LIN {X 0,Y 569.864,Z 352.293,A -85,B 0,C 180,E1 27134.007,E2 27134.007} C_VEL
LIN {X 0,Y 571.953,Z 355.251,A -85,B 0,C 180,E1 27133.743,E2 27133.743} C_VEL
LIN {X 0,Y 584.357,Z 373.532,A -85,B 0,C 180,E1 27132.228,E2 27132.228} C_VEL
LIN {X 0,Y 595.034,Z 390.48,A -85,B 0,C 180,E1 27130.982,E2 27130.982} C_VEL
LIN {X 0,Y 605.418,Z 407.827,A -85,B 0,C 180,E1 27129.82,E2 27129.82} C_VEL
LIN {X 0,Y 601.344,Z 587.031,A -85,B 0,C 180,E1 27127.412,E2 27127.412} C_VEL
LIN {X 0,Y 600.399,Z 594.727,A -85,B 0,C 180,E1 27127.369,E2 27127.369} C_VEL
LIN {X 0,Y 595.054,Z 615.267,A -85,B 0,C 180,E1 27127.472,E2 27127.472} C_VEL
LIN {X 0,Y 594.323,Z 621.871,A -85,B 0,C 180,E1 27127.429,E2 27127.429} C_VEL
LIN {X 0,Y 591.491,Z 740.275,A -85,B 0,C 180,E1 27125.822,E2 27125.822} C_VEL
LIN {X 0,Y 590.199,Z 765.933,A -85,B 0,C 180,E1 27125.308,E2 27125.308} C_VEL
LIN {X 0,Y 588.778,Z 786.603,A -85,B 0,C 180,E1 27124.752,E2 27124.752} C_VEL
LIN {X 0,Y 586.911,Z 809.672,A -85,B 0,C 180,E1 27123.973,E2 27123.973} C_VEL
LIN {X 0,Y 584.739,Z 831.447,A -85,B 0,C 180,E1 27123.058,E2 27123.058} C_VEL
LIN {X 0,Y 582.598,Z 851.106,A -85,B 0,C 180,E1 27122.085,E2 27122.085} C_VEL
LIN {X 0,Y 579.921,Z 873.043,A -85,B 0,C 180,E1 27120.803,E2 27120.803} C_VEL
LIN {X 0,Y 577.554,Z 891.278,A -85,B 0,C 180,E1 27119.565,E2 27119.565} C_VEL
LIN {X 0,Y 574.708,Z 912.427,A -85,B 0,C 180,E1 27117.905,E2 27117.905} C_VEL
LIN {X 0,Y 572.362,Z 929.084,A -85,B 0,C 180,E1 27116.398,E2 27116.398} C_VEL
LIN {X 0,Y 569.881,Z 946.877,A -85,B 0,C 180,E1 27114.572,E2 27114.572} C_VEL
LIN {X 0,Y 567.593,Z 963.267,A -85,B 0,C 180,E1 27112.616,E2 27112.616} C_VEL
LIN {X 0,Y 565.641,Z 978.22,A -85,B 0,C 180,E1 27110.596,E2 27110.596} C_VEL
LIN {X 0,Y 563.908,Z 992.141,A -85,B 0,C 180,E1 27108.398,E2 27108.398} C_VEL
LIN {X 0,Y 562.601,Z 1004.328,A -85,B 0,C 180,E1 27106.202,E2 27106.202} C_VEL
LIN {X 0,Y 561.55,Z 1015.061,A -85,B 0,C 180,E1 27103.909,E2 27103.909} C_VEL
LIN {X 0,Y 560.865,Z 1023.83,A -85,B 0,C 180,E1 27101.726,E2 27101.726} C_VEL
LIN {X 0,Y 560.352,Z 1032.037,A -85,B 0,C 180,E1 27099.241,E2 27099.241} C_VEL
LIN {X 0,Y 560.1,Z 1037.791,A -85,B 0,C 180,E1 27097.076,E2 27097.076} C_VEL
LIN {X 0,Y 559.965,Z 1042.874,A -85,B 0,C 180,E1 27094.609,E2 27094.609} C_VEL
LIN {X 0,Y 559.925,Z 1046.117,A -85,B 0,C 180,E1 27092.252,E2 27092.252} C_VEL
LIN {X 0,Y 559.918,Z 1047.976,A -85,B 0,C 180,E1 27090,E2 27090} C_VEL
LIN {X 0,Y 559.896,Z 1048.458,A -85,B 0,C 180,E1 27087.441,E2 27087.441} C_VEL
LIN {X 0,Y 559.901,Z 1047.57,A -85,B 0,C 180,E1 27085.288,E2 27085.288} C_VEL
LIN {X 0,Y 559.937,Z 1045.192,A -85,B 0,C 180,E1 27082.819,E2 27082.819} C_VEL
LIN {X 0,Y 559.998,Z 1041.245,A -85,B 0,C 180,E1 27080.442,E2 27080.442} C_VEL
LIN {X 0,Y 560.165,Z 1036.402,A -85,B 0,C 180,E1 27078.259,E2 27078.259} C_VEL
LIN {X 0,Y 560.544,Z 1028.866,A -85,B 0,C 180,E1 27075.644,E2 27075.644} C_VEL
LIN {X 0,Y 561.057,Z 1021.218,A -85,B 0,C 180,E1 27073.497,E2 27073.497} C_VEL
LIN {X 0,Y 561.93,Z 1011.097,A -85,B 0,C 180,E1 27071.104,E2 27071.104} C_VEL
LIN {X 0,Y 562.978,Z 1000.415,A -85,B 0,C 180,E1 27068.976,E2 27068.976} C_VEL
LIN {X 0,Y 564.484,Z 987.53,A -85,B 0,C 180,E1 27066.734,E2 27066.734} C_VEL
LIN {X 0,Y 566.302,Z 973.067,A -85,B 0,C 180,E1 27064.593,E2 27064.593} C_VEL
LIN {X 0,Y 568.423,Z 957.461,A -85,B 0,C 180,E1 27062.557,E2 27062.557} C_VEL
LIN {X 0,Y 570.744,Z 940.758,A -85,B 0,C 180,E1 27060.682,E2 27060.682} C_VEL
LIN {X 0,Y 573.203,Z 923.555,A -85,B 0,C 180,E1 27058.971,E2 27058.971} C_VEL
LIN {X 0,Y 575.887,Z 904.313,A -85,B 0,C 180,E1 27057.318,E2 27057.318} C_VEL
LIN {X 0,Y 578.42,Z 885.955,A -85,B 0,C 180,E1 27055.938,E2 27055.938} C_VEL
LIN {X 0,Y 581.277,Z 863.847,A -85,B 0,C 180,E1 27054.51,E2 27054.51} C_VEL
LIN {X 0,Y 583.53,Z 844.808,A -85,B 0,C 180,E1 27053.457,E2 27053.457} C_VEL
LIN {X 0,Y 585.978,Z 822.583,A -85,B 0,C 180,E1 27052.409,E2 27052.409} C_VEL
LIN {X 0,Y 588.031,Z 800.135,A -85,B 0,C 180,E1 27051.543,E2 27051.543} C_VEL
LIN {X 0,Y 589.972,Z 776.277,A -85,B 0,C 180,E1 27050.802,E2 27050.802} C_VEL
LIN {X 0,Y 591.358,Z 753.251,A -85,B 0,C 180,E1 27050.269,E2 27050.269} C_VEL
LIN {X 0,Y 592.323,Z 730.378,A -85,B 0,C 180,E1 27049.878,E2 27049.878} C_VEL
LIN {X 0,Y 598.539,Z 477.791,A -85,B 0,C 180,E1 27046.449,E2 27046.449} C_VEL
LIN {X 0,Y 600.073,Z 410.838,A -85,B 0,C 180,E1 27045.512,E2 27045.512} C_VEL
LIN {X 0,Y 587.214,Z 389.608,A -85,B 0,C 180,E1 27043.955,E2 27043.955} C_VEL
LIN {X 0,Y 573.32,Z 368.918,A -85,B 0,C 180,E1 27042.18,E2 27042.18} C_VEL
LIN {X 0,Y 567.731,Z 361.268,A -85,B 0,C 180,E1 27041.435,E2 27041.435} C_VEL
LIN {X 0,Y 564.464,Z 356.623,A -85,B 0,C 180,E1 27040.985,E2 27040.985} C_VEL
LIN {X 0,Y 562.218,Z 353.874,A -85,B 0,C 180,E1 27040.679,E2 27040.679} C_VEL
LIN {X 0,Y 561.563,Z 351.979,A -85,B 0,C 180,E1 27040.534,E2 27040.534} C_VEL
LIN {X 0,Y 561.445,Z 351.25,A -85,B 0,C 180,E1 27040.411,E2 27040.411} C_VEL
LIN {X 0,Y 561.381,Z 351.276,A -85,B 0,C 180,E1 27037.235,E2 27037.235} C_VEL
LIN {X 0,Y 561.417,Z 351.281,A -85,B 0,C 180,E1 27033.906,E2 27033.906} C_VEL
LIN {X 0,Y 561.401,Z 351.292,A -85,B 0,C 180,E1 27030.742,E2 27030.742} C_VEL
LIN {X 0,Y 561.387,Z 351.299,A -85,B 0,C 180,E1 27027.357,E2 27027.357} C_VEL
LIN {X 0,Y 561.441,Z 351.289,A -85,B 0,C 180,E1 27024.181,E2 27024.181} C_VEL
LIN {X 0,Y 561.381,Z 351.291,A -85,B 0,C 180,E1 27020.978,E2 27020.978} C_VEL
LIN {X 0,Y 561.424,Z 351.283,A -85,B 0,C 180,E1 27017.731,E2 27017.731} C_VEL
LIN {X 0,Y 561.386,Z 351.293,A -85,B 0,C 180,E1 27014.65,E2 27014.65} C_VEL
LIN {X 0,Y 561.389,Z 351.296,A -85,B 0,C 180,E1 27011.195,E2 27011.195} C_VEL
LIN {X 0,Y 561.437,Z 351.298,A -85,B 0,C 180,E1 27007.985,E2 27007.985} C_VEL
LIN {X 0,Y 561.379,Z 351.292,A -85,B 0,C 180,E1 27004.802,E2 27004.802} C_VEL
LIN {X 0,Y 561.433,Z 351.279,A -85,B 0,C 180,E1 27001.531,E2 27001.531} C_VEL
LIN {X 0,Y 561.384,Z 351.301,A -85,B 0,C 180,E1 26998.469,E2 26998.469} C_VEL
LIN {X 0,Y 561.4,Z 351.299,A -85,B 0,C 180,E1 26995.096,E2 26995.096} C_VEL
LIN {X 0,Y 561.401,Z 351.285,A -85,B 0,C 180,E1 26992.014,E2 26992.014} C_VEL
LIN {X 0,Y 561.38,Z 351.281,A -85,B 0,C 180,E1 26988.701,E2 26988.701} C_VEL
LIN {X 0,Y 561.448,Z 351.281,A -85,B 0,C 180,E1 26985.457,E2 26985.457} C_VEL
LIN {X 0,Y 561.382,Z 351.3,A -85,B 0,C 180,E1 26982.267,E2 26982.267} C_VEL
LIN {X 0,Y 561.412,Z 351.298,A -85,B 0,C 180,E1 26978.948,E2 26978.948} C_VEL
LIN {X 0,Y 561.388,Z 351.287,A -85,B 0,C 180,E1 26975.929,E2 26975.929} C_VEL
LIN {X 0,Y 561.386,Z 351.288,A -85,B 0,C 180,E1 26972.498,E2 26972.498} C_VEL
LIN {X 0,Y 561.419,Z 351.3,A -85,B 0,C 180,E1 26969.497,E2 26969.497} C_VEL
LIN {X 0,Y 561.38,Z 351.303,A -85,B 0,C 180,E1 26966.24,E2 26966.24} C_VEL
LIN {X 0,Y 561.441,Z 351.299,A -85,B 0,C 180,E1 26962.99,E2 26962.99} C_VEL
LIN {X 0,Y 561.382,Z 351.304,A -85,B 0,C 180,E1 26959.827,E2 26959.827} C_VEL
LIN {X 0,Y 561.555,Z 352.203,A -85,B 0,C 180,E1 26959.648,E2 26959.648} C_VEL
LIN {X 0,Y 563.435,Z 356.303,A -85,B 0,C 180,E1 26958.957,E2 26958.957} C_VEL
LIN {X 0,Y 569.718,Z 370.71,A -85,B 0,C 180,E1 26956.667,E2 26956.667} C_VEL
LIN {X 0,Y 570.766,Z 373.125,A -85,B 0,C 180,E1 26956.352,E2 26956.352} C_VEL
LIN {X 0,Y 582.747,Z 391.401,A -85,B 0,C 180,E1 26954.789,E2 26954.789} C_VEL
LIN {X 0,Y 595.371,Z 412.407,A -85,B 0,C 180,E1 26953.225,E2 26953.225} C_VEL
LIN {X 0,Y 600.003,Z 420.961,A -85,B 0,C 180,E1 26952.664,E2 26952.664} C_VEL
LIN {X 0,Y 600.16,Z 425.019,A -85,B 0,C 180,E1 26952.585,E2 26952.585} C_VEL
LIN {X 0,Y 593.701,Z 685.414,A -85,B 0,C 180,E1 26949.041,E2 26949.041} C_VEL
LIN {X 0,Y 591.65,Z 766.034,A -85,B 0,C 180,E1 26947.933,E2 26947.933} C_VEL
LIN {X 0,Y 590.187,Z 791.581,A -85,B 0,C 180,E1 26947.422,E2 26947.422} C_VEL
LIN {X 0,Y 588.579,Z 813.335,A -85,B 0,C 180,E1 26946.836,E2 26946.836} C_VEL
LIN {X 0,Y 586.38,Z 838.196,A -85,B 0,C 180,E1 26945.975,E2 26945.975} C_VEL
LIN {X 0,Y 584.287,Z 858.471,A -85,B 0,C 180,E1 26945.114,E2 26945.114} C_VEL
LIN {X 0,Y 581.811,Z 880.444,A -85,B 0,C 180,E1 26944.014,E2 26944.014} C_VEL
LIN {X 0,Y 579.215,Z 901.047,A -85,B 0,C 180,E1 26942.785,E2 26942.785} C_VEL
LIN {X 0,Y 576.615,Z 921.114,A -85,B 0,C 180,E1 26941.411,E2 26941.411} C_VEL
LIN {X 0,Y 573.894,Z 941.134,A -85,B 0,C 180,E1 26939.812,E2 26939.812} C_VEL
LIN {X 0,Y 571.553,Z 958.312,A -85,B 0,C 180,E1 26938.252,E2 26938.252} C_VEL
LIN {X 0,Y 568.994,Z 977.194,A -85,B 0,C 180,E1 26936.285,E2 26936.285} C_VEL
LIN {X 0,Y 567.016,Z 992.376,A -85,B 0,C 180,E1 26934.482,E2 26934.482} C_VEL
LIN {X 0,Y 564.997,Z 1008.815,A -85,B 0,C 180,E1 26932.245,E2 26932.245} C_VEL
LIN {X 0,Y 563.613,Z 1020.97,A -85,B 0,C 180,E1 26930.348,E2 26930.348} C_VEL
LIN {X 0,Y 562.316,Z 1034.002,A -85,B 0,C 180,E1 26928.023,E2 26928.023} C_VEL
LIN {X 0,Y 561.398,Z 1044.512,A -85,B 0,C 180,E1 26925.813,E2 26925.813} C_VEL
LIN {X 0,Y 560.745,Z 1053.948,A -85,B 0,C 180,E1 26923.509,E2 26923.509} C_VEL
LIN {X 0,Y 560.304,Z 1061.89,A -85,B 0,C 180,E1 26921.112,E2 26921.112} C_VEL
LIN {X 0,Y 560.065,Z 1067.774,A -85,B 0,C 180,E1 26918.935,E2 26918.935} C_VEL
LIN {X 0,Y 559.949,Z 1073.035,A -85,B 0,C 180,E1 26916.356,E2 26916.356} C_VEL
LIN {X 0,Y 559.914,Z 1076.033,A -85,B 0,C 180,E1 26914.199,E2 26914.199} C_VEL
LIN {X 0,Y 559.904,Z 1077.913,A -85,B 0,C 180,E1 26911.944,E2 26911.944} C_VEL
LIN {X 0,Y 559.896,Z 1078.345,A -85,B 0,C 180,E1 26909.488,E2 26909.488} C_VEL
LIN {X 0,Y 559.907,Z 1077.429,A -85,B 0,C 180,E1 26907.339,E2 26907.339} C_VEL
LIN {X 0,Y 559.931,Z 1075.107,A -85,B 0,C 180,E1 26904.98,E2 26904.98} C_VEL
LIN {X 0,Y 559.984,Z 1070.929,A -85,B 0,C 180,E1 26902.51,E2 26902.51} C_VEL
LIN {X 0,Y 560.134,Z 1066.227,A -85,B 0,C 180,E1 26900.444,E2 26900.444} C_VEL
LIN {X 0,Y 560.464,Z 1058.71,A -85,B 0,C 180,E1 26897.866,E2 26897.866} C_VEL
LIN {X 0,Y 560.952,Z 1050.667,A -85,B 0,C 180,E1 26895.655,E2 26895.655} C_VEL
LIN {X 0,Y 561.76,Z 1040.359,A -85,B 0,C 180,E1 26893.257,E2 26893.257} C_VEL
LIN {X 0,Y 562.796,Z 1028.901,A -85,B 0,C 180,E1 26891.027,E2 26891.027} C_VEL
LIN {X 0,Y 564.22,Z 1015.654,A -85,B 0,C 180,E1 26888.775,E2 26888.775} C_VEL
LIN {X 0,Y 565.906,Z 1001.267,A -85,B 0,C 180,E1 26886.685,E2 26886.685} C_VEL
LIN {X 0,Y 567.913,Z 985.575,A -85,B 0,C 180,E1 26884.67,E2 26884.67} C_VEL
LIN {X 0,Y 570.192,Z 968.342,A -85,B 0,C 180,E1 26882.758,E2 26882.758} C_VEL
LIN {X 0,Y 572.443,Z 951.643,A -85,B 0,C 180,E1 26881.121,E2 26881.121} C_VEL
LIN {X 0,Y 575.208,Z 931.042,A -85,B 0,C 180,E1 26879.369,E2 26879.369} C_VEL
LIN {X 0,Y 577.627,Z 912.745,A -85,B 0,C 180,E1 26878.015,E2 26878.015} C_VEL
LIN {X 0,Y 580.49,Z 889.767,A -85,B 0,C 180,E1 26876.551,E2 26876.551} C_VEL
LIN {X 0,Y 582.689,Z 870.64,A -85,B 0,C 180,E1 26875.509,E2 26875.509} C_VEL
LIN {X 0,Y 585.179,Z 847.637,A -85,B 0,C 180,E1 26874.445,E2 26874.445} C_VEL
LIN {X 0,Y 587.18,Z 825.79,A -85,B 0,C 180,E1 26873.619,E2 26873.619} C_VEL
LIN {X 0,Y 589.127,Z 802.224,A -85,B 0,C 180,E1 26872.895,E2 26872.895} C_VEL
LIN {X 0,Y 590.595,Z 778.451,A -85,B 0,C 180,E1 26872.352,E2 26872.352} C_VEL
LIN {X 0,Y 591.556,Z 755.977,A -85,B 0,C 180,E1 26871.973,E2 26871.973} C_VEL
LIN {X 0,Y 597.259,Z 507.123,A -85,B 0,C 180,E1 26868.626,E2 26868.626} C_VEL
LIN {X 0,Y 599.18,Z 421.264,A -85,B 0,C 180,E1 26867.448,E2 26867.448} C_VEL
LIN {X 0,Y 598.222,Z 418.74,A -85,B 0,C 180,E1 26867.326,E2 26867.326} C_VEL
LIN {X 0,Y 584.047,Z 394.647,A -85,B 0,C 180,E1 26865.677,E2 26865.677} C_VEL
LIN {X 0,Y 570.279,Z 372.684,A -85,B 0,C 180,E1 26863.973,E2 26863.973} C_VEL
LIN {X 0,Y 564.417,Z 358.728,A -85,B 0,C 180,E1 26861.903,E2 26861.903} C_VEL
LIN {X 0,Y 561.425,Z 351.294,A -85,B 0,C 180,E1 26860.743,E2 26860.743} C_VEL
LIN {X 0,Y 561.384,Z 351.292,A -85,B 0,C 180,E1 26857.656,E2 26857.656} C_VEL
LIN {X 0,Y 561.388,Z 351.287,A -85,B 0,C 180,E1 26854.252,E2 26854.252} C_VEL
LIN {X 0,Y 561.409,Z 351.284,A -85,B 0,C 180,E1 26851.217,E2 26851.217} C_VEL
LIN {X 0,Y 561.381,Z 351.287,A -85,B 0,C 180,E1 26847.933,E2 26847.933} C_VEL
LIN {X 0,Y 561.443,Z 351.291,A -85,B 0,C 180,E1 26844.732,E2 26844.732} C_VEL
LIN {X 0,Y 561.38,Z 351.299,A -85,B 0,C 180,E1 26841.525,E2 26841.525} C_VEL
LIN {X 0,Y 561.414,Z 351.282,A -85,B 0,C 180,E1 26838.268,E2 26838.268} C_VEL
LIN {X 0,Y 561.395,Z 351.288,A -85,B 0,C 180,E1 26835.128,E2 26835.128} C_VEL
LIN {X 0,Y 561.389,Z 351.3,A -85,B 0,C 180,E1 26831.819,E2 26831.819} C_VEL
LIN {X 0,Y 561.435,Z 351.276,A -85,B 0,C 180,E1 26828.604,E2 26828.604} C_VEL
LIN {X 0,Y 561.379,Z 351.288,A -85,B 0,C 180,E1 26825.417,E2 26825.417} C_VEL
LIN {X 0,Y 561.432,Z 351.297,A -85,B 0,C 180,E1 26822.143,E2 26822.143} C_VEL
LIN {X 0,Y 561.381,Z 351.274,A -85,B 0,C 180,E1 26819.081,E2 26819.081} C_VEL
LIN {X 0,Y 561.399,Z 351.293,A -85,B 0,C 180,E1 26815.71,E2 26815.71} C_VEL
LIN {X 0,Y 561.405,Z 351.288,A -85,B 0,C 180,E1 26812.632,E2 26812.632} C_VEL
LIN {X 0,Y 561.382,Z 351.278,A -85,B 0,C 180,E1 26809.325,E2 26809.325} C_VEL
LIN {X 0,Y 561.45,Z 351.297,A -85,B 0,C 180,E1 26806.07,E2 26806.07} C_VEL
LIN {X 0,Y 561.382,Z 351.29,A -85,B 0,C 180,E1 26802.909,E2 26802.909} C_VEL
LIN {X 0,Y 561.424,Z 351.279,A -85,B 0,C 180,E1 26799.678,E2 26799.678} C_VEL
LIN {X 0,Y 561.392,Z 351.299,A -85,B 0,C 180,E1 26796.598,E2 26796.598} C_VEL
LIN {X 0,Y 561.393,Z 351.3,A -85,B 0,C 180,E1 26793.167,E2 26793.167} C_VEL
LIN {X 0,Y 561.425,Z 351.278,A -85,B 0,C 180,E1 26790.087,E2 26790.087} C_VEL
LIN {X 0,Y 561.382,Z 351.284,A -85,B 0,C 180,E1 26786.838,E2 26786.838} C_VEL
LIN {X 0,Y 561.44,Z 351.284,A -85,B 0,C 180,E1 26783.609,E2 26783.609} C_VEL
LIN {X 0,Y 561.385,Z 351.292,A -85,B 0,C 180,E1 26780.464,E2 26780.464} C_VEL
LIN {X 0,Y 561.413,Z 351.266,A -85,B 0,C 180,E1 26777.204,E2 26777.204} C_VEL
LIN {X 0,Y 561.416,Z 351.4,A -85,B 0,C 180,E1 26774.971,E2 26774.971} C_VEL
LIN {X 0,Y 561.764,Z 352.877,A -85,B 0,C 180,E1 26774.84,E2 26774.84} C_VEL
LIN {X 0,Y 563.667,Z 355.936,A -85,B 0,C 180,E1 26774.584,E2 26774.584} C_VEL
LIN {X 0,Y 565.182,Z 357.543,A -85,B 0,C 180,E1 26774.396,E2 26774.396} C_VEL
LIN {X 0,Y 567.902,Z 361.521,A -85,B 0,C 180,E1 26774.045,E2 26774.045} C_VEL
LIN {X 0,Y 579.907,Z 379.342,A -85,B 0,C 180,E1 26772.551,E2 26772.551} C_VEL
LIN {X 0,Y 590.434,Z 396.155,A -85,B 0,C 180,E1 26771.299,E2 26771.299} C_VEL
LIN {X 0,Y 599.337,Z 411.062,A -85,B 0,C 180,E1 26770.282,E2 26770.282} C_VEL
LIN {X 0,Y 594.323,Z 621.871,A -85,B 0,C 180,E1 26767.429,E2 26767.429} C_VEL
LIN {X 0,Y 593.377,Z 629.565,A -85,B 0,C 180,E1 26767.385,E2 26767.385} C_VEL
LIN {X 0,Y 588.018,Z 650.1,A -85,B 0,C 180,E1 26767.491,E2 26767.491} C_VEL
LIN {X 0,Y 587.273,Z 656.704,A -85,B 0,C 180,E1 26767.448,E2 26767.448} C_VEL
LIN {X 0,Y 585.108,Z 741.247,A -85,B 0,C 180,E1 26766.284,E2 26766.284} C_VEL
LIN {X 0,Y 583.771,Z 766.42,A -85,B 0,C 180,E1 26765.771,E2 26765.771} C_VEL
LIN {X 0,Y 582.282,Z 787.179,A -85,B 0,C 180,E1 26765.207,E2 26765.207} C_VEL
LIN {X 0,Y 580.17,Z 811.758,A -85,B 0,C 180,E1 26764.357,E2 26764.357} C_VEL
LIN {X 0,Y 578.055,Z 832.103,A -85,B 0,C 180,E1 26763.49,E2 26763.49} C_VEL
LIN {X 0,Y 575.616,Z 853.587,A -85,B 0,C 180,E1 26762.411,E2 26762.411} C_VEL
LIN {X 0,Y 572.808,Z 875.188,A -85,B 0,C 180,E1 26761.111,E2 26761.111} C_VEL
LIN {X 0,Y 570.082,Z 895.415,A -85,B 0,C 180,E1 26759.702,E2 26759.702} C_VEL
LIN {X 0,Y 567.3,Z 914.704,A -85,B 0,C 180,E1 26758.13,E2 26758.13} C_VEL
LIN {X 0,Y 564.872,Z 931.192,A -85,B 0,C 180,E1 26756.605,E2 26756.605} C_VEL
LIN {X 0,Y 562.083,Z 950.048,A -85,B 0,C 180,E1 26754.599,E2 26754.599} C_VEL
LIN {X 0,Y 559.944,Z 964.791,A -85,B 0,C 180,E1 26752.799,E2 26752.799} C_VEL
LIN {X 0,Y 557.643,Z 981.381,A -85,B 0,C 180,E1 26750.466,E2 26750.466} C_VEL
LIN {X 0,Y 556.042,Z 993.781,A -85,B 0,C 180,E1 26748.451,E2 26748.451} C_VEL
LIN {X 0,Y 554.51,Z 1007.231,A -85,B 0,C 180,E1 26745.908,E2 26745.908} C_VEL
LIN {X 0,Y 553.567,Z 1016.753,A -85,B 0,C 180,E1 26743.794,E2 26743.794} C_VEL
LIN {X 0,Y 552.795,Z 1026.378,A -85,B 0,C 180,E1 26741.265,E2 26741.265} C_VEL
LIN {X 0,Y 552.35,Z 1033.227,A -85,B 0,C 180,E1 26739.061,E2 26739.061} C_VEL
LIN {X 0,Y 552.085,Z 1039.323,A -85,B 0,C 180,E1 26736.656,E2 26736.656} C_VEL
LIN {X 0,Y 551.964,Z 1043.913,A -85,B 0,C 180,E1 26734.155,E2 26734.155} C_VEL
LIN {X 0,Y 551.926,Z 1046.697,A -85,B 0,C 180,E1 26731.973,E2 26731.973} C_VEL
LIN {X 0,Y 551.907,Z 1048.478,A -85,B 0,C 180,E1 26729.377,E2 26729.377} C_VEL
LIN {X 0,Y 551.906,Z 1048.598,A -85,B 0,C 180,E1 26727.092,E2 26727.092} C_VEL
LIN {X 0,Y 551.915,Z 1047.498,A -85,B 0,C 180,E1 26724.803,E2 26724.803} C_VEL
LIN {X 0,Y 551.945,Z 1044.574,A -85,B 0,C 180,E1 26722.191,E2 26722.191} C_VEL
LIN {X 0,Y 552.022,Z 1040.994,A -85,B 0,C 180,E1 26720.091,E2 26720.091} C_VEL
LIN {X 0,Y 552.247,Z 1035.536,A -85,B 0,C 180,E1 26717.664,E2 26717.664} C_VEL
LIN {X 0,Y 552.659,Z 1028.281,A -85,B 0,C 180,E1 26715.22,E2 26715.22} C_VEL
LIN {X 0,Y 553.283,Z 1020.145,A -85,B 0,C 180,E1 26712.943,E2 26712.943} C_VEL
LIN {X 0,Y 554.253,Z 1009.629,A -85,B 0,C 180,E1 26710.504,E2 26710.504} C_VEL
LIN {X 0,Y 555.467,Z 998.753,A -85,B 0,C 180,E1 26708.345,E2 26708.345} C_VEL
LIN {X 0,Y 557.208,Z 984.751,A -85,B 0,C 180,E1 26705.962,E2 26705.962} C_VEL
LIN {X 0,Y 559.009,Z 971.523,A -85,B 0,C 180,E1 26704.009,E2 26704.009} C_VEL
LIN {X 0,Y 561.449,Z 954.593,A -85,B 0,C 180,E1 26701.831,E2 26701.831} C_VEL
LIN {X 0,Y 563.739,Z 939.212,A -85,B 0,C 180,E1 26700.106,E2 26700.106} C_VEL
LIN {X 0,Y 566.545,Z 920.579,A -85,B 0,C 180,E1 26698.269,E2 26698.269} C_VEL
LIN {X 0,Y 569.193,Z 902.626,A -85,B 0,C 180,E1 26696.739,E2 26696.739} C_VEL
LIN {X 0,Y 572.136,Z 882.347,A -85,B 0,C 180,E1 26695.225,E2 26695.225} C_VEL
LIN {X 0,Y 574.829,Z 861.887,A -85,B 0,C 180,E1 26693.928,E2 26693.928} C_VEL
LIN {X 0,Y 577.425,Z 840.954,A -85,B 0,C 180,E1 26692.78,E2 26692.78} C_VEL
LIN {X 0,Y 579.913,Z 818.416,A -85,B 0,C 180,E1 26691.758,E2 26691.758} C_VEL
LIN {X 0,Y 581.859,Z 798.04,A -85,B 0,C 180,E1 26690.985,E2 26690.985} C_VEL
LIN {X 0,Y 583.902,Z 772.802,A -85,B 0,C 180,E1 26690.227,E2 26690.227} C_VEL
LIN {X 0,Y 585.175,Z 752.148,A -85,B 0,C 180,E1 26689.756,E2 26689.756} C_VEL
LIN {X 0,Y 586.212,Z 727.492,A -85,B 0,C 180,E1 26689.342,E2 26689.342} C_VEL
LIN {X 0,Y 592.735,Z 474.327,A -85,B 0,C 180,E1 26685.878,E2 26685.878} C_VEL
LIN {X 0,Y 594.185,Z 414.117,A -85,B 0,C 180,E1 26685.027,E2 26685.027} C_VEL
LIN {X 0,Y 580.889,Z 392.482,A -85,B 0,C 180,E1 26683.378,E2 26683.378} C_VEL
LIN {X 0,Y 568.738,Z 374.274,A -85,B 0,C 180,E1 26681.784,E2 26681.784} C_VEL
LIN {X 0,Y 563.794,Z 367.478,A -85,B 0,C 180,E1 26681.112,E2 26681.112} C_VEL
LIN {X 0,Y 560.388,Z 362.809,A -85,B 0,C 180,E1 26680.637,E2 26680.637} C_VEL
LIN {X 0,Y 557.686,Z 358.97,A -85,B 0,C 180,E1 26680.25,E2 26680.25} C_VEL
LIN {X 0,Y 556.886,Z 357.84,A -85,B 0,C 180,E1 26680.135,E2 26680.135} C_VEL
LIN {X 0,Y 554.43,Z 355.202,A -85,B 0,C 180,E1 26679.792,E2 26679.792} C_VEL
LIN {X 0,Y 553.443,Z 352.256,A -85,B 0,C 180,E1 26679.574,E2 26679.574} C_VEL
LIN {X 0,Y 553.49,Z 352.239,A -85,B 0,C 180,E1 26676.466,E2 26676.466} C_VEL
LIN {X 0,Y 553.443,Z 352.291,A -85,B 0,C 180,E1 26673.191,E2 26673.191} C_VEL
LIN {X 0,Y 553.484,Z 352.286,A -85,B 0,C 180,E1 26669.872,E2 26669.872} C_VEL
LIN {X 0,Y 553.454,Z 352.29,A -85,B 0,C 180,E1 26666.814,E2 26666.814} C_VEL
LIN {X 0,Y 553.452,Z 352.289,A -85,B 0,C 180,E1 26663.397,E2 26663.397} C_VEL
LIN {X 0,Y 553.488,Z 352.282,A -85,B 0,C 180,E1 26660.295,E2 26660.295} C_VEL
LIN {X 0,Y 553.441,Z 352.282,A -85,B 0,C 180,E1 26657.019,E2 26657.019} C_VEL
LIN {X 0,Y 553.5,Z 352.269,A -85,B 0,C 180,E1 26653.796,E2 26653.796} C_VEL
LIN {X 0,Y 553.446,Z 352.281,A -85,B 0,C 180,E1 26650.619,E2 26650.619} C_VEL
LIN {X 0,Y 553.451,Z 352.286,A -85,B 0,C 180,E1 26647.161,E2 26647.161} C_VEL
LIN {X 0,Y 553.492,Z 352.285,A -85,B 0,C 180,E1 26643.936,E2 26643.936} C_VEL
LIN {X 0,Y 553.439,Z 352.277,A -85,B 0,C 180,E1 26640.725,E2 26640.725} C_VEL
LIN {X 0,Y 553.494,Z 352.267,A -85,B 0,C 180,E1 26637.515,E2 26637.515} C_VEL
LIN {X 0,Y 553.448,Z 352.291,A -85,B 0,C 180,E1 26634.297,E2 26634.297} C_VEL
LIN {X 0,Y 553.449,Z 352.288,A -85,B 0,C 180,E1 26630.852,E2 26630.852} C_VEL
LIN {X 0,Y 553.498,Z 352.273,A -85,B 0,C 180,E1 26627.586,E2 26627.586} C_VEL
LIN {X 0,Y 553.439,Z 352.27,A -85,B 0,C 180,E1 26624.357,E2 26624.357} C_VEL
LIN {X 0,Y 553.485,Z 352.268,A -85,B 0,C 180,E1 26621.133,E2 26621.133} C_VEL
LIN {X 0,Y 553.453,Z 352.287,A -85,B 0,C 180,E1 26617.942,E2 26617.942} C_VEL
LIN {X 0,Y 553.447,Z 352.289,A -85,B 0,C 180,E1 26614.533,E2 26614.533} C_VEL
LIN {X 0,Y 553.509,Z 352.286,A -85,B 0,C 180,E1 26611.281,E2 26611.281} C_VEL
LIN {X 0,Y 553.44,Z 352.29,A -85,B 0,C 180,E1 26608.118,E2 26608.118} C_VEL
LIN {X 0,Y 553.483,Z 352.288,A -85,B 0,C 180,E1 26604.81,E2 26604.81} C_VEL
LIN {X 0,Y 553.454,Z 352.291,A -85,B 0,C 180,E1 26601.636,E2 26601.636} C_VEL
LIN {X 0,Y 553.479,Z 352.358,A -85,B 0,C 180,E1 26600.616,E2 26600.616} C_VEL
LIN {X 0,Y 554.665,Z 355.655,A -85,B 0,C 180,E1 26600.077,E2 26600.077} C_VEL
LIN {X 0,Y 558.806,Z 364.624,A -85,B 0,C 180,E1 26598.543,E2 26598.543} C_VEL
LIN {X 0,Y 562.281,Z 372.587,A -85,B 0,C 180,E1 26597.297,E2 26597.297} C_VEL
LIN {X 0,Y 574.651,Z 391.348,A -85,B 0,C 180,E1 26595.615,E2 26595.615} C_VEL
LIN {X 0,Y 587.888,Z 412.893,A -85,B 0,C 180,E1 26593.921,E2 26593.921} C_VEL
LIN {X 0,Y 594.346,Z 424.545,A -85,B 0,C 180,E1 26593.121,E2 26593.121} C_VEL
LIN {X 0,Y 587.538,Z 685.487,A -85,B 0,C 180,E1 26589.538,E2 26589.538} C_VEL
LIN {X 0,Y 585.395,Z 765.84,A -85,B 0,C 180,E1 26588.423,E2 26588.423} C_VEL
LIN {X 0,Y 583.856,Z 791.505,A -85,B 0,C 180,E1 26587.907,E2 26587.907} C_VEL
LIN {X 0,Y 582.157,Z 813.446,A -85,B 0,C 180,E1 26587.311,E2 26587.311} C_VEL
LIN {X 0,Y 579.857,Z 838.217,A -85,B 0,C 180,E1 26586.445,E2 26586.445} C_VEL
LIN {X 0,Y 577.731,Z 857.924,A -85,B 0,C 180,E1 26585.601,E2 26585.601} C_VEL
LIN {X 0,Y 575.077,Z 880.382,A -85,B 0,C 180,E1 26584.468,E2 26584.468} C_VEL
LIN {X 0,Y 572.309,Z 901.331,A -85,B 0,C 180,E1 26583.205,E2 26583.205} C_VEL
LIN {X 0,Y 569.514,Z 921.819,A -85,B 0,C 180,E1 26581.783,E2 26581.783} C_VEL
LIN {X 0,Y 566.635,Z 941.805,A -85,B 0,C 180,E1 26580.156,E2 26580.156} C_VEL
LIN {X 0,Y 564.042,Z 959.907,A -85,B 0,C 180,E1 26578.481,E2 26578.481} C_VEL
LIN {X 0,Y 561.436,Z 977.937,A -85,B 0,C 180,E1 26576.553,E2 26576.553} C_VEL
LIN {X 0,Y 559.365,Z 993.012,A -85,B 0,C 180,E1 26574.726,E2 26574.726} C_VEL
LIN {X 0,Y 557.245,Z 1009.251,A -85,B 0,C 180,E1 26572.468,E2 26572.468} C_VEL
LIN {X 0,Y 555.717,Z 1022.031,A -85,B 0,C 180,E1 26570.43,E2 26570.43} C_VEL
LIN {X 0,Y 554.313,Z 1035.345,A -85,B 0,C 180,E1 26567.966,E2 26567.966} C_VEL
LIN {X 0,Y 553.459,Z 1044.756,A -85,B 0,C 180,E1 26565.939,E2 26565.939} C_VEL
LIN {X 0,Y 552.749,Z 1054.477,A -85,B 0,C 180,E1 26563.495,E2 26563.495} C_VEL
LIN {X 0,Y 552.313,Z 1061.979,A -85,B 0,C 180,E1 26561.169,E2 26561.169} C_VEL
LIN {X 0,Y 552.061,Z 1068.073,A -85,B 0,C 180,E1 26558.856,E2 26558.856} C_VEL
LIN {X 0,Y 551.95,Z 1072.982,A -85,B 0,C 180,E1 26556.344,E2 26556.344} C_VEL
LIN {X 0,Y 551.916,Z 1075.818,A -85,B 0,C 180,E1 26554.26,E2 26554.26} C_VEL
LIN {X 0,Y 551.907,Z 1077.7,A -85,B 0,C 180,E1 26551.973,E2 26551.973} C_VEL
LIN {X 0,Y 551.899,Z 1078.132,A -85,B 0,C 180,E1 26549.481,E2 26549.481} C_VEL
LIN {X 0,Y 551.91,Z 1077.216,A -85,B 0,C 180,E1 26547.3,E2 26547.3} C_VEL
LIN {X 0,Y 551.933,Z 1074.893,A -85,B 0,C 180,E1 26544.907,E2 26544.907} C_VEL
LIN {X 0,Y 551.985,Z 1070.925,A -85,B 0,C 180,E1 26542.506,E2 26542.506} C_VEL
LIN {X 0,Y 552.143,Z 1066.011,A -85,B 0,C 180,E1 26540.304,E2 26540.304} C_VEL
LIN {X 0,Y 552.484,Z 1058.767,A -85,B 0,C 180,E1 26537.769,E2 26537.769} C_VEL
LIN {X 0,Y 552.991,Z 1050.86,A -85,B 0,C 180,E1 26535.551,E2 26535.551} C_VEL
LIN {X 0,Y 553.802,Z 1041.052,A -85,B 0,C 180,E1 26533.209,E2 26533.209} C_VEL
LIN {X 0,Y 554.932,Z 1029.263,A -85,B 0,C 180,E1 26530.857,E2 26530.857} C_VEL
LIN {X 0,Y 556.317,Z 1016.916,A -85,B 0,C 180,E1 26528.712,E2 26528.712} C_VEL
LIN {X 0,Y 558.197,Z 1001.827,A -85,B 0,C 180,E1 26526.456,E2 26526.456} C_VEL
LIN {X 0,Y 560.083,Z 987.69,A -85,B 0,C 180,E1 26524.601,E2 26524.601} C_VEL
LIN {X 0,Y 562.679,Z 969.137,A -85,B 0,C 180,E1 26522.482,E2 26522.482} C_VEL
LIN {X 0,Y 564.952,Z 953.042,A -85,B 0,C 180,E1 26520.875,E2 26520.875} C_VEL
LIN {X 0,Y 567.91,Z 932.216,A -85,B 0,C 180,E1 26519.062,E2 26519.062} C_VEL
LIN {X 0,Y 570.445,Z 913.895,A -85,B 0,C 180,E1 26517.682,E2 26517.682} C_VEL
LIN {X 0,Y 573.323,Z 892.216,A -85,B 0,C 180,E1 26516.263,E2 26516.263} C_VEL
LIN {X 0,Y 575.838,Z 871.262,A -85,B 0,C 180,E1 26515.1,E2 26515.1} C_VEL
LIN {X 0,Y 578.364,Z 849.264,A -85,B 0,C 180,E1 26514.06,E2 26514.06} C_VEL
LIN {X 0,Y 580.57,Z 826.283,A -85,B 0,C 180,E1 26513.177,E2 26513.177} C_VEL
LIN {X 0,Y 582.501,Z 803.812,A -85,B 0,C 180,E1 26512.475,E2 26512.475} C_VEL
LIN {X 0,Y 584.13,Z 779.377,A -85,B 0,C 180,E1 26511.9,E2 26511.9} C_VEL
LIN {X 0,Y 585.129,Z 757.488,A -85,B 0,C 180,E1 26511.522,E2 26511.522} C_VEL
LIN {X 0,Y 591.025,Z 513.048,A -85,B 0,C 180,E1 26508.202,E2 26508.202} C_VEL
LIN {X 0,Y 593.157,Z 423.688,A -85,B 0,C 180,E1 26506.968,E2 26506.968} C_VEL
LIN {X 0,Y 578.927,Z 399.379,A -85,B 0,C 180,E1 26505.276,E2 26505.276} C_VEL
LIN {X 0,Y 565.486,Z 377.953,A -85,B 0,C 180,E1 26503.581,E2 26503.581} C_VEL
LIN {X 0,Y 561.718,Z 372.03,A -85,B 0,C 180,E1 26503.052,E2 26503.052} C_VEL
LIN {X 0,Y 554.96,Z 356.032,A -85,B 0,C 180,E1 26500.574,E2 26500.574} C_VEL
LIN {X 0,Y 553.473,Z 352.517,A -85,B 0,C 180,E1 26500.005,E2 26500.005} C_VEL
LIN {X 0,Y 553.493,Z 352.272,A -85,B 0,C 180,E1 26497.112,E2 26497.112} C_VEL
LIN {X 0,Y 553.44,Z 352.278,A -85,B 0,C 180,E1 26493.811,E2 26493.811} C_VEL
LIN {X 0,Y 553.479,Z 352.271,A -85,B 0,C 180,E1 26490.507,E2 26490.507} C_VEL
LIN {X 0,Y 553.448,Z 352.27,A -85,B 0,C 180,E1 26487.432,E2 26487.432} C_VEL
LIN {X 0,Y 553.445,Z 352.273,A -85,B 0,C 180,E1 26483.985,E2 26483.985} C_VEL
LIN {X 0,Y 553.496,Z 352.286,A -85,B 0,C 180,E1 26480.848,E2 26480.848} C_VEL
LIN {X 0,Y 553.441,Z 352.287,A -85,B 0,C 180,E1 26477.561,E2 26477.561} C_VEL
LIN {X 0,Y 553.491,Z 352.264,A -85,B 0,C 180,E1 26474.329,E2 26474.329} C_VEL
LIN {X 0,Y 553.452,Z 352.286,A -85,B 0,C 180,E1 26471.146,E2 26471.146} C_VEL
LIN {X 0,Y 553.447,Z 352.29,A -85,B 0,C 180,E1 26467.683,E2 26467.683} C_VEL
LIN {X 0,Y 553.49,Z 352.262,A -85,B 0,C 180,E1 26464.559,E2 26464.559} C_VEL
LIN {X 0,Y 553.441,Z 352.288,A -85,B 0,C 180,E1 26461.346,E2 26461.346} C_VEL
LIN {X 0,Y 553.496,Z 352.266,A -85,B 0,C 180,E1 26458.137,E2 26458.137} C_VEL
LIN {X 0,Y 553.448,Z 352.277,A -85,B 0,C 180,E1 26454.921,E2 26454.921} C_VEL
LIN {X 0,Y 553.451,Z 352.29,A -85,B 0,C 180,E1 26451.481,E2 26451.481} C_VEL
LIN {X 0,Y 553.495,Z 352.26,A -85,B 0,C 180,E1 26448.221,E2 26448.221} C_VEL
LIN {X 0,Y 553.442,Z 352.281,A -85,B 0,C 180,E1 26445.027,E2 26445.027} C_VEL
LIN {X 0,Y 553.493,Z 352.285,A -85,B 0,C 180,E1 26441.788,E2 26441.788} C_VEL
LIN {X 0,Y 553.452,Z 352.269,A -85,B 0,C 180,E1 26438.596,E2 26438.596} C_VEL
LIN {X 0,Y 553.453,Z 352.27,A -85,B 0,C 180,E1 26435.22,E2 26435.22} C_VEL
LIN {X 0,Y 553.502,Z 352.284,A -85,B 0,C 180,E1 26431.986,E2 26431.986} C_VEL
LIN {X 0,Y 553.446,Z 352.29,A -85,B 0,C 180,E1 26428.767,E2 26428.767} C_VEL
LIN {X 0,Y 553.487,Z 352.281,A -85,B 0,C 180,E1 26425.465,E2 26425.465} C_VEL
LIN {X 0,Y 553.461,Z 352.285,A -85,B 0,C 180,E1 26422.233,E2 26422.233} C_VEL
LIN {X 0,Y 553.453,Z 352.292,A -85,B 0,C 180,E1 26418.881,E2 26418.881} C_VEL
LIN {X 0,Y 553.516,Z 352.422,A -85,B 0,C 180,E1 26415.747,E2 26415.747} C_VEL
LIN {X 0,Y 554.737,Z 355.613,A -85,B 0,C 180,E1 26415.552,E2 26415.552} C_VEL
LIN {X 0,Y 557.304,Z 358.568,A -85,B 0,C 180,E1 26415.216,E2 26415.216} C_VEL
LIN {X 0,Y 560.041,Z 362.58,A -85,B 0,C 180,E1 26414.848,E2 26414.848} C_VEL
LIN {X 0,Y 567.608,Z 373.212,A -85,B 0,C 180,E1 26413.868,E2 26413.868} C_VEL
LIN {X 0,Y 581.618,Z 394.667,A -85,B 0,C 180,E1 26412.132,E2 26412.132} C_VEL
LIN {X 0,Y 593.291,Z 414.33,A -85,B 0,C 180,E1 26410.753,E2 26410.753} C_VEL
LIN {X 0,Y 587.273,Z 656.704,A -85,B 0,C 180,E1 26407.448,E2 26407.448} C_VEL
LIN {X 0,Y 586.31,Z 664.399,A -85,B 0,C 180,E1 26407.405,E2 26407.405} C_VEL
LIN {X 0,Y 580.934,Z 684.929,A -85,B 0,C 180,E1 26407.514,E2 26407.514} C_VEL
LIN {X 0,Y 580.191,Z 691.532,A -85,B 0,C 180,E1 26407.47,E2 26407.47} C_VEL
LIN {X 0,Y 578.713,Z 743.986,A -85,B 0,C 180,E1 26406.727,E2 26406.727} C_VEL
LIN {X 0,Y 577.312,Z 767.92,A -85,B 0,C 180,E1 26406.219,E2 26406.219} C_VEL
LIN {X 0,Y 575.729,Z 789.042,A -85,B 0,C 180,E1 26405.633,E2 26405.633} C_VEL
LIN {X 0,Y 573.476,Z 813.615,A -85,B 0,C 180,E1 26404.76,E2 26404.76} C_VEL
LIN {X 0,Y 571.275,Z 833.863,A -85,B 0,C 180,E1 26403.88,E2 26403.88} C_VEL
LIN {X 0,Y 568.599,Z 856.085,A -85,B 0,C 180,E1 26402.734,E2 26402.734} C_VEL
LIN {X 0,Y 565.934,Z 875.723,A -85,B 0,C 180,E1 26401.532,E2 26401.532} C_VEL
LIN {X 0,Y 562.986,Z 896.638,A -85,B 0,C 180,E1 26400.056,E2 26400.056} C_VEL
LIN {X 0,Y 560.079,Z 915.772,A -85,B 0,C 180,E1 26398.468,E2 26398.468} C_VEL
LIN {X 0,Y 557.469,Z 932.739,A -85,B 0,C 180,E1 26396.872,E2 26396.872} C_VEL
LIN {X 0,Y 554.693,Z 950.508,A -85,B 0,C 180,E1 26394.945,E2 26394.945} C_VEL
LIN {X 0,Y 552.453,Z 965.214,A -85,B 0,C 180,E1 26393.126,E2 26393.126} C_VEL
LIN {X 0,Y 550.12,Z 981.104,A -85,B 0,C 180,E1 26390.87,E2 26390.87} C_VEL
LIN {X 0,Y 548.462,Z 993.237,A -85,B 0,C 180,E1 26388.882,E2 26388.882} C_VEL
LIN {X 0,Y 546.884,Z 1006.084,A -85,B 0,C 180,E1 26386.463,E2 26386.463} C_VEL
LIN {X 0,Y 545.776,Z 1016.202,A -85,B 0,C 180,E1 26384.211,E2 26384.211} C_VEL
LIN {X 0,Y 544.95,Z 1025.658,A -85,B 0,C 180,E1 26381.751,E2 26381.751} C_VEL
LIN {X 0,Y 544.408,Z 1033.231,A -85,B 0,C 180,E1 26379.301,E2 26379.301} C_VEL
LIN {X 0,Y 544.119,Z 1039.11,A -85,B 0,C 180,E1 26376.966,E2 26376.966} C_VEL
LIN {X 0,Y 543.975,Z 1043.859,A -85,B 0,C 180,E1 26374.428,E2 26374.428} C_VEL
LIN {X 0,Y 543.935,Z 1046.719,A -85,B 0,C 180,E1 26372.212,E2 26372.212} C_VEL
LIN {X 0,Y 543.91,Z 1048.63,A -85,B 0,C 180,E1 26369.684,E2 26369.684} C_VEL
LIN {X 0,Y 543.904,Z 1048.85,A -85,B 0,C 180,E1 26367.26,E2 26367.26} C_VEL
LIN {X 0,Y 543.911,Z 1047.945,A -85,B 0,C 180,E1 26365.125,E2 26365.125} C_VEL
LIN {X 0,Y 543.943,Z 1045.533,A -85,B 0,C 180,E1 26362.607,E2 26362.607} C_VEL
LIN {X 0,Y 544.029,Z 1041.559,A -85,B 0,C 180,E1 26360.158,E2 26360.158} C_VEL
LIN {X 0,Y 544.229,Z 1036.691,A -85,B 0,C 180,E1 26357.91,E2 26357.91} C_VEL
LIN {X 0,Y 544.667,Z 1029.45,A -85,B 0,C 180,E1 26355.325,E2 26355.325} C_VEL
LIN {X 0,Y 545.249,Z 1021.983,A -85,B 0,C 180,E1 26353.157,E2 26353.157} C_VEL
LIN {X 0,Y 546.21,Z 1012.263,A -85,B 0,C 180,E1 26350.761,E2 26350.761} C_VEL
LIN {X 0,Y 547.47,Z 1001.093,A -85,B 0,C 180,E1 26348.463,E2 26348.463} C_VEL
LIN {X 0,Y 549.156,Z 988.247,A -85,B 0,C 180,E1 26346.158,E2 26346.158} C_VEL
LIN {X 0,Y 551.198,Z 973.856,A -85,B 0,C 180,E1 26343.96,E2 26343.96} C_VEL
LIN {X 0,Y 553.43,Z 959.175,A -85,B 0,C 180,E1 26341.982,E2 26341.982} C_VEL
LIN {X 0,Y 556.081,Z 942.25,A -85,B 0,C 180,E1 26340.008,E2 26340.008} C_VEL
LIN {X 0,Y 558.6,Z 926.284,A -85,B 0,C 180,E1 26338.368,E2 26338.368} C_VEL
LIN {X 0,Y 561.851,Z 905.525,A -85,B 0,C 180,E1 26336.517,E2 26336.517} C_VEL
LIN {X 0,Y 564.509,Z 887.997,A -85,B 0,C 180,E1 26335.164,E2 26335.164} C_VEL
LIN {X 0,Y 567.634,Z 866.271,A -85,B 0,C 180,E1 26333.711,E2 26333.711} C_VEL
LIN {X 0,Y 570.163,Z 846.787,A -85,B 0,C 180,E1 26332.601,E2 26332.601} C_VEL
LIN {X 0,Y 572.736,Z 825.719,A -85,B 0,C 180,E1 26331.574,E2 26331.574} C_VEL
LIN {X 0,Y 575.102,Z 802.41,A -85,B 0,C 180,E1 26330.642,E2 26330.642} C_VEL
LIN {X 0,Y 577.063,Z 780.294,A -85,B 0,C 180,E1 26329.927,E2 26329.927} C_VEL
LIN {X 0,Y 578.78,Z 755.543,A -85,B 0,C 180,E1 26329.321,E2 26329.321} C_VEL
LIN {X 0,Y 579.816,Z 733.707,A -85,B 0,C 180,E1 26328.932,E2 26328.932} C_VEL
LIN {X 0,Y 586.618,Z 484.146,A -85,B 0,C 180,E1 26325.48,E2 26325.48} C_VEL
LIN {X 0,Y 588.402,Z 417.526,A -85,B 0,C 180,E1 26324.54,E2 26324.54} C_VEL
LIN {X 0,Y 575.019,Z 395.806,A -85,B 0,C 180,E1 26322.836,E2 26322.836} C_VEL
LIN {X 0,Y 561.085,Z 375.029,A -85,B 0,C 180,E1 26320.947,E2 26320.947} C_VEL
LIN {X 0,Y 553.737,Z 365.162,A -85,B 0,C 180,E1 26319.903,E2 26319.903} C_VEL
LIN {X 0,Y 550.099,Z 360.585,A -85,B 0,C 180,E1 26319.373,E2 26319.373} C_VEL
LIN {X 0,Y 549.271,Z 359.092,A -85,B 0,C 180,E1 26319.242,E2 26319.242} C_VEL
LIN {X 0,Y 546.699,Z 356.549,A -85,B 0,C 180,E1 26318.871,E2 26318.871} C_VEL
LIN {X 0,Y 545.557,Z 353.379,A -85,B 0,C 180,E1 26318.663,E2 26318.663} C_VEL
LIN {X 0,Y 545.5,Z 353.228,A -85,B 0,C 180,E1 26315.346,E2 26315.346} C_VEL
LIN {X 0,Y 545.56,Z 353.263,A -85,B 0,C 180,E1 26312.107,E2 26312.107} C_VEL
LIN {X 0,Y 545.51,Z 353.27,A -85,B 0,C 180,E1 26308.94,E2 26308.94} C_VEL
LIN {X 0,Y 545.517,Z 353.264,A -85,B 0,C 180,E1 26305.514,E2 26305.514} C_VEL
LIN {X 0,Y 545.558,Z 353.262,A -85,B 0,C 180,E1 26302.248,E2 26302.248} C_VEL
LIN {X 0,Y 545.507,Z 353.276,A -85,B 0,C 180,E1 26298.949,E2 26298.949} C_VEL
LIN {X 0,Y 545.541,Z 353.274,A -85,B 0,C 180,E1 26295.63,E2 26295.63} C_VEL
LIN {X 0,Y 545.517,Z 353.274,A -85,B 0,C 180,E1 26292.491,E2 26292.491} C_VEL
LIN {X 0,Y 545.506,Z 353.269,A -85,B 0,C 180,E1 26289.07,E2 26289.07} C_VEL
LIN {X 0,Y 545.561,Z 353.256,A -85,B 0,C 180,E1 26285.891,E2 26285.891} C_VEL
LIN {X 0,Y 545.504,Z 353.277,A -85,B 0,C 180,E1 26282.606,E2 26282.606} C_VEL
LIN {X 0,Y 545.533,Z 353.276,A -85,B 0,C 180,E1 26279.265,E2 26279.265} C_VEL
LIN {X 0,Y 545.532,Z 353.266,A -85,B 0,C 180,E1 26276.006,E2 26276.006} C_VEL
LIN {X 0,Y 545.502,Z 353.258,A -85,B 0,C 180,E1 26272.734,E2 26272.734} C_VEL
LIN {X 0,Y 545.559,Z 353.259,A -85,B 0,C 180,E1 26269.546,E2 26269.546} C_VEL
LIN {X 0,Y 545.504,Z 353.279,A -85,B 0,C 180,E1 26266.281,E2 26266.281} C_VEL
LIN {X 0,Y 545.528,Z 353.275,A -85,B 0,C 180,E1 26262.947,E2 26262.947} C_VEL
LIN {X 0,Y 545.531,Z 353.26,A -85,B 0,C 180,E1 26259.732,E2 26259.732} C_VEL
LIN {X 0,Y 545.502,Z 353.26,A -85,B 0,C 180,E1 26256.447,E2 26256.447} C_VEL
LIN {X 0,Y 545.562,Z 353.256,A -85,B 0,C 180,E1 26253.197,E2 26253.197} C_VEL
LIN {X 0,Y 545.503,Z 353.277,A -85,B 0,C 180,E1 26250.095,E2 26250.095} C_VEL
LIN {X 0,Y 545.538,Z 353.275,A -85,B 0,C 180,E1 26246.768,E2 26246.768} C_VEL
LIN {X 0,Y 545.522,Z 353.277,A -85,B 0,C 180,E1 26243.568,E2 26243.568} C_VEL
LIN {X 0,Y 545.547,Z 353.434,A -85,B 0,C 180,E1 26241.501,E2 26241.501} C_VEL
LIN {X 0,Y 546.943,Z 356.866,A -85,B 0,C 180,E1 26240.897,E2 26240.897} C_VEL
LIN {X 0,Y 552.731,Z 369.791,A -85,B 0,C 180,E1 26238.654,E2 26238.654} C_VEL
LIN {X 0,Y 553.923,Z 372.421,A -85,B 0,C 180,E1 26238.269,E2 26238.269} C_VEL
LIN {X 0,Y 566.29,Z 390.72,A -85,B 0,C 180,E1 26236.517,E2 26236.517} C_VEL
LIN {X 0,Y 578.478,Z 410.325,A -85,B 0,C 180,E1 26234.89,E2 26234.89} C_VEL
LIN {X 0,Y 588.478,Z 427.51,A -85,B 0,C 180,E1 26233.62,E2 26233.62} C_VEL
LIN {X 0,Y 581.414,Z 685.931,A -85,B 0,C 180,E1 26230.041,E2 26230.041} C_VEL
LIN {X 0,Y 579.185,Z 765.672,A -85,B 0,C 180,E1 26228.924,E2 26228.924} C_VEL
LIN {X 0,Y 577.58,Z 791.315,A -85,B 0,C 180,E1 26228.405,E2 26228.405} C_VEL
LIN {X 0,Y 575.8,Z 813.335,A -85,B 0,C 180,E1 26227.803,E2 26227.803} C_VEL
LIN {X 0,Y 573.376,Z 838.25,A -85,B 0,C 180,E1 26226.924,E2 26226.924} C_VEL
LIN {X 0,Y 571.195,Z 857.607,A -85,B 0,C 180,E1 26226.09,E2 26226.09} C_VEL
LIN {X 0,Y 568.389,Z 880.253,A -85,B 0,C 180,E1 26224.938,E2 26224.938} C_VEL
LIN {X 0,Y 565.532,Z 900.948,A -85,B 0,C 180,E1 26223.678,E2 26223.678} C_VEL
LIN {X 0,Y 562.652,Z 920.988,A -85,B 0,C 180,E1 26222.277,E2 26222.277} C_VEL
LIN {X 0,Y 559.666,Z 940.68,A -85,B 0,C 180,E1 26220.668,E2 26220.668} C_VEL
LIN {X 0,Y 557.039,Z 958.054,A -85,B 0,C 180,E1 26219.053,E2 26219.053} C_VEL
LIN {X 0,Y 554.171,Z 976.838,A -85,B 0,C 180,E1 26217.045,E2 26217.045} C_VEL
LIN {X 0,Y 551.96,Z 991.974,A -85,B 0,C 180,E1 26215.196,E2 26215.196} C_VEL
LIN {X 0,Y 549.686,Z 1008.315,A -85,B 0,C 180,E1 26212.909,E2 26212.909} C_VEL
LIN {X 0,Y 548.05,Z 1021.164,A -85,B 0,C 180,E1 26210.841,E2 26210.841} C_VEL
LIN {X 0,Y 546.494,Z 1034.945,A -85,B 0,C 180,E1 26208.27,E2 26208.27} C_VEL
LIN {X 0,Y 545.565,Z 1044.534,A -85,B 0,C 180,E1 26206.175,E2 26206.175} C_VEL
LIN {X 0,Y 544.805,Z 1054.257,A -85,B 0,C 180,E1 26203.695,E2 26203.695} C_VEL
LIN {X 0,Y 544.338,Z 1061.76,A -85,B 0,C 180,E1 26201.335,E2 26201.335} C_VEL
LIN {X 0,Y 544.07,Z 1067.856,A -85,B 0,C 180,E1 26198.987,E2 26198.987} C_VEL
LIN {X 0,Y 543.949,Z 1072.766,A -85,B 0,C 180,E1 26196.438,E2 26196.438} C_VEL
LIN {X 0,Y 543.918,Z 1075.604,A -85,B 0,C 180,E1 26194.323,E2 26194.323} C_VEL
LIN {X 0,Y 543.91,Z 1077.486,A -85,B 0,C 180,E1 26192.002,E2 26192.002} C_VEL
LIN {X 0,Y 543.902,Z 1077.918,A -85,B 0,C 180,E1 26189.473,E2 26189.473} C_VEL
LIN {X 0,Y 543.912,Z 1077.003,A -85,B 0,C 180,E1 26187.26,E2 26187.26} C_VEL
LIN {X 0,Y 543.934,Z 1074.679,A -85,B 0,C 180,E1 26184.832,E2 26184.832} C_VEL
LIN {X 0,Y 543.986,Z 1070.71,A -85,B 0,C 180,E1 26182.395,E2 26182.395} C_VEL
LIN {X 0,Y 544.145,Z 1066.055,A -85,B 0,C 180,E1 26180.267,E2 26180.267} C_VEL
LIN {X 0,Y 544.484,Z 1059.287,A -85,B 0,C 180,E1 26177.808,E2 26177.808} C_VEL
LIN {X 0,Y 545.031,Z 1051.054,A -85,B 0,C 180,E1 26175.444,E2 26175.444} C_VEL
LIN {X 0,Y 545.787,Z 1042.23,A -85,B 0,C 180,E1 26173.284,E2 26173.284} C_VEL
LIN {X 0,Y 547.007,Z 1030.206,A -85,B 0,C 180,E1 26170.79,E2 26170.79} C_VEL
LIN {X 0,Y 548.367,Z 1018.548,A -85,B 0,C 180,E1 26168.711,E2 26168.711} C_VEL
LIN {X 0,Y 550.294,Z 1003.93,A -85,B 0,C 180,E1 26166.438,E2 26166.438} C_VEL
LIN {X 0,Y 552.309,Z 989.361,A -85,B 0,C 180,E1 26164.477,E2 26164.477} C_VEL
LIN {X 0,Y 554.838,Z 972.333,A -85,B 0,C 180,E1 26162.456,E2 26162.456} C_VEL
LIN {X 0,Y 557.462,Z 954.481,A -85,B 0,C 180,E1 26160.628,E2 26160.628} C_VEL
LIN {X 0,Y 560.362,Z 935.264,A -85,B 0,C 180,E1 26158.897,E2 26158.897} C_VEL
LIN {X 0,Y 563.173,Z 915.778,A -85,B 0,C 180,E1 26157.395,E2 26157.395} C_VEL
LIN {X 0,Y 565.83,Z 896.882,A -85,B 0,C 180,E1 26156.115,E2 26156.115} C_VEL
LIN {X 0,Y 568.774,Z 873.901,A -85,B 0,C 180,E1 26154.787,E2 26154.787} C_VEL
LIN {X 0,Y 571.274,Z 853.014,A -85,B 0,C 180,E1 26153.77,E2 26153.77} C_VEL
LIN {X 0,Y 573.845,Z 828.285,A -85,B 0,C 180,E1 26152.778,E2 26152.778} C_VEL
LIN {X 0,Y 575.738,Z 807.183,A -85,B 0,C 180,E1 26152.098,E2 26152.098} C_VEL
LIN {X 0,Y 577.644,Z 781.289,A -85,B 0,C 180,E1 26151.458,E2 26151.458} C_VEL
LIN {X 0,Y 578.728,Z 759.201,A -85,B 0,C 180,E1 26151.065,E2 26151.065} C_VEL
LIN {X 0,Y 584.791,Z 520.135,A -85,B 0,C 180,E1 26147.786,E2 26147.786} C_VEL
LIN {X 0,Y 587.154,Z 426.916,A -85,B 0,C 180,E1 26146.489,E2 26146.489} C_VEL
LIN {X 0,Y 571.809,Z 400.651,A -85,B 0,C 180,E1 26144.612,E2 26144.612} C_VEL
LIN {X 0,Y 559.047,Z 380.64,A -85,B 0,C 180,E1 26142.957,E2 26142.957} C_VEL
LIN {X 0,Y 553.395,Z 371.842,A -85,B 0,C 180,E1 26142.163,E2 26142.163} C_VEL
LIN {X 0,Y 548.431,Z 360.447,A -85,B 0,C 180,E1 26140.333,E2 26140.333} C_VEL
LIN {X 0,Y 545.613,Z 353.686,A -85,B 0,C 180,E1 26139.216,E2 26139.216} C_VEL
LIN {X 0,Y 545.563,Z 353.268,A -85,B 0,C 180,E1 26139.085,E2 26139.085} C_VEL
LIN {X 0,Y 545.503,Z 353.282,A -85,B 0,C 180,E1 26135.783,E2 26135.783} C_VEL
LIN {X 0,Y 545.533,Z 353.276,A -85,B 0,C 180,E1 26132.482,E2 26132.482} C_VEL
LIN {X 0,Y 545.517,Z 353.275,A -85,B 0,C 180,E1 26129.421,E2 26129.421} C_VEL
LIN {X 0,Y 545.507,Z 353.274,A -85,B 0,C 180,E1 26125.981,E2 26125.981} C_VEL
LIN {X 0,Y 545.567,Z 353.251,A -85,B 0,C 180,E1 26122.75,E2 26122.75} C_VEL
LIN {X 0,Y 545.502,Z 353.261,A -85,B 0,C 180,E1 26119.488,E2 26119.488} C_VEL
LIN {X 0,Y 545.531,Z 353.274,A -85,B 0,C 180,E1 26116.173,E2 26116.173} C_VEL
LIN {X 0,Y 545.522,Z 353.268,A -85,B 0,C 180,E1 26113.029,E2 26113.029} C_VEL
LIN {X 0,Y 545.505,Z 353.253,A -85,B 0,C 180,E1 26109.708,E2 26109.708} C_VEL
LIN {X 0,Y 545.571,Z 353.272,A -85,B 0,C 180,E1 26106.419,E2 26106.419} C_VEL
LIN {X 0,Y 545.505,Z 353.27,A -85,B 0,C 180,E1 26103.152,E2 26103.152} C_VEL
LIN {X 0,Y 545.521,Z 353.252,A -85,B 0,C 180,E1 26099.79,E2 26099.79} C_VEL
LIN {X 0,Y 545.534,Z 353.275,A -85,B 0,C 180,E1 26096.638,E2 26096.638} C_VEL
LIN {X 0,Y 545.504,Z 353.259,A -85,B 0,C 180,E1 26093.369,E2 26093.369} C_VEL
LIN {X 0,Y 545.561,Z 353.262,A -85,B 0,C 180,E1 26090.186,E2 26090.186} C_VEL
LIN {X 0,Y 545.509,Z 353.276,A -85,B 0,C 180,E1 26086.863,E2 26086.863} C_VEL
LIN {X 0,Y 545.519,Z 353.257,A -85,B 0,C 180,E1 26083.459,E2 26083.459} C_VEL
LIN {X 0,Y 545.545,Z 353.267,A -85,B 0,C 180,E1 26080.291,E2 26080.291} C_VEL
LIN {X 0,Y 545.508,Z 353.279,A -85,B 0,C 180,E1 26077.019,E2 26077.019} C_VEL
LIN {X 0,Y 545.562,Z 353.255,A -85,B 0,C 180,E1 26073.788,E2 26073.788} C_VEL
LIN {X 0,Y 545.51,Z 353.258,A -85,B 0,C 180,E1 26070.578,E2 26070.578} C_VEL
LIN {X 0,Y 545.518,Z 353.261,A -85,B 0,C 180,E1 26067.143,E2 26067.143} C_VEL
LIN {X 0,Y 545.552,Z 353.265,A -85,B 0,C 180,E1 26063.927,E2 26063.927} C_VEL
LIN {X 0,Y 545.505,Z 353.271,A -85,B 0,C 180,E1 26060.639,E2 26060.639} C_VEL
LIN {X 0,Y 545.556,Z 353.244,A -85,B 0,C 180,E1 26057.445,E2 26057.445} C_VEL
LIN {X 0,Y 545.524,Z 353.391,A -85,B 0,C 180,E1 26056.64,E2 26056.64} C_VEL
LIN {X 0,Y 546.695,Z 356.539,A -85,B 0,C 180,E1 26056.444,E2 26056.444} C_VEL
LIN {X 0,Y 549.535,Z 359.67,A -85,B 0,C 180,E1 26056.059,E2 26056.059} C_VEL
LIN {X 0,Y 552.166,Z 363.52,A -85,B 0,C 180,E1 26055.69,E2 26055.69} C_VEL
LIN {X 0,Y 562.945,Z 378.525,A -85,B 0,C 180,E1 26054.254,E2 26054.254} C_VEL
LIN {X 0,Y 577.16,Z 400.506,A -85,B 0,C 180,E1 26052.455,E2 26052.455} C_VEL
LIN {X 0,Y 587.285,Z 417.698,A -85,B 0,C 180,E1 26051.232,E2 26051.232} C_VEL
LIN {X 0,Y 580.842,Z 665.424,A -85,B 0,C 180,E1 26047.826,E2 26047.826} C_VEL
LIN {X 0,Y 580.191,Z 691.532,A -85,B 0,C 180,E1 26047.47,E2 26047.47} C_VEL
LIN {X 0,Y 579.237,Z 699.223,A -85,B 0,C 180,E1 26047.426,E2 26047.426} C_VEL
LIN {X 0,Y 573.858,Z 719.75,A -85,B 0,C 180,E1 26047.537,E2 26047.537} C_VEL
LIN {X 0,Y 573.08,Z 726.354,A -85,B 0,C 180,E1 26047.495,E2 26047.495} C_VEL
LIN {X 0,Y 572.003,Z 751.824,A -85,B 0,C 180,E1 26047.071,E2 26047.071} C_VEL
LIN {X 0,Y 570.686,Z 772.366,A -85,B 0,C 180,E1 26046.602,E2 26046.602} C_VEL
LIN {X 0,Y 568.636,Z 797.064,A -85,B 0,C 180,E1 26045.863,E2 26045.863} C_VEL
LIN {X 0,Y 566.572,Z 817.66,A -85,B 0,C 180,E1 26045.083,E2 26045.083} C_VEL
LIN {X 0,Y 564.003,Z 840.035,A -85,B 0,C 180,E1 26044.071,E2 26044.071} C_VEL
LIN {X 0,Y 561.11,Z 861.963,A -85,B 0,C 180,E1 26042.862,E2 26042.862} C_VEL
LIN {X 0,Y 558.208,Z 882.64,A -85,B 0,C 180,E1 26041.537,E2 26041.537} C_VEL
LIN {X 0,Y 555.065,Z 903.039,A -85,B 0,C 180,E1 26039.992,E2 26039.992} C_VEL
LIN {X 0,Y 552.221,Z 921.02,A -85,B 0,C 180,E1 26038.438,E2 26038.438} C_VEL
LIN {X 0,Y 549.207,Z 939.328,A -85,B 0,C 180,E1 26036.607,E2 26036.607} C_VEL
LIN {X 0,Y 546.755,Z 954.528,A -85,B 0,C 180,E1 26034.874,E2 26034.874} C_VEL
LIN {X 0,Y 543.979,Z 971.939,A -85,B 0,C 180,E1 26032.592,E2 26032.592} C_VEL
LIN {X 0,Y 542.016,Z 984.923,A -85,B 0,C 180,E1 26030.631,E2 26030.631} C_VEL
LIN {X 0,Y 539.993,Z 999.294,A -85,B 0,C 180,E1 26028.124,E2 26028.124} C_VEL
LIN {X 0,Y 538.655,Z 1010.001,A -85,B 0,C 180,E1 26025.939,E2 26025.939} C_VEL
LIN {X 0,Y 537.499,Z 1020.862,A -85,B 0,C 180,E1 26023.337,E2 26023.337} C_VEL
LIN {X 0,Y 536.808,Z 1028.736,A -85,B 0,C 180,E1 26021.061,E2 26021.061} C_VEL
LIN {X 0,Y 536.338,Z 1035.901,A -85,B 0,C 180,E1 26018.577,E2 26018.577} C_VEL
LIN {X 0,Y 536.068,Z 1041.325,A -85,B 0,C 180,E1 26016.103,E2 26016.103} C_VEL
LIN {X 0,Y 535.965,Z 1045.057,A -85,B 0,C 180,E1 26013.851,E2 26013.851} C_VEL
LIN {X 0,Y 535.926,Z 1047.938,A -85,B 0,C 180,E1 26011.176,E2 26011.176} C_VEL
LIN {X 0,Y 535.915,Z 1049.006,A -85,B 0,C 180,E1 26008.931,E2 26008.931} C_VEL
LIN {X 0,Y 535.915,Z 1048.946,A -85,B 0,C 180,E1 26006.684,E2 26006.684} C_VEL
LIN {X 0,Y 535.937,Z 1047.259,A -85,B 0,C 180,E1 26003.943,E2 26003.943} C_VEL
LIN {X 0,Y 535.982,Z 1044.441,A -85,B 0,C 180,E1 26001.633,E2 26001.633} C_VEL
LIN {X 0,Y 536.119,Z 1040.085,A -85,B 0,C 180,E1 25999.142,E2 25999.142} C_VEL
LIN {X 0,Y 536.43,Z 1034.004,A -85,B 0,C 180,E1 25996.636,E2 25996.636} C_VEL
LIN {X 0,Y 536.937,Z 1027.114,A -85,B 0,C 180,E1 25994.335,E2 25994.335} C_VEL
LIN {X 0,Y 537.836,Z 1017.399,A -85,B 0,C 180,E1 25991.688,E2 25991.688} C_VEL
LIN {X 0,Y 538.943,Z 1007.721,A -85,B 0,C 180,E1 25989.473,E2 25989.473} C_VEL
LIN {X 0,Y 540.651,Z 994.638,A -85,B 0,C 180,E1 25986.916,E2 25986.916} C_VEL
LIN {X 0,Y 542.438,Z 982.245,A -85,B 0,C 180,E1 25984.834,E2 25984.834} C_VEL
LIN {X 0,Y 544.874,Z 966.806,A -85,B 0,C 180,E1 25982.574,E2 25982.574} C_VEL
LIN {X 0,Y 547.286,Z 951.914,A -85,B 0,C 180,E1 25980.683,E2 25980.683} C_VEL
LIN {X 0,Y 550.212,Z 934.606,A -85,B 0,C 180,E1 25978.746,E2 25978.746} C_VEL
LIN {X 0,Y 553.189,Z 916.48,A -85,B 0,C 180,E1 25977.002,E2 25977.002} C_VEL
LIN {X 0,Y 556.389,Z 896.896,A -85,B 0,C 180,E1 25975.346,E2 25975.346} C_VEL
LIN {X 0,Y 559.532,Z 876.209,A -85,B 0,C 180,E1 25973.863,E2 25973.863} C_VEL
LIN {X 0,Y 562.581,Z 855.295,A -85,B 0,C 180,E1 25972.566,E2 25972.566} C_VEL
LIN {X 0,Y 565.399,Z 833.348,A -85,B 0,C 180,E1 25971.43,E2 25971.43} C_VEL
LIN {X 0,Y 567.648,Z 814.001,A -85,B 0,C 180,E1 25970.579,E2 25970.579} C_VEL
LIN {X 0,Y 570.061,Z 789.555,A -85,B 0,C 180,E1 25969.699,E2 25969.699} C_VEL
LIN {X 0,Y 571.773,Z 768.263,A -85,B 0,C 180,E1 25969.1,E2 25969.1} C_VEL
LIN {X 0,Y 573.277,Z 744.413,A -85,B 0,C 180,E1 25968.587,E2 25968.587} C_VEL
LIN {X 0,Y 574.895,Z 692.081,A -85,B 0,C 180,E1 25967.833,E2 25967.833} C_VEL
LIN {X 0,Y 582.054,Z 442.595,A -85,B 0,C 180,E1 25964.352,E2 25964.352} C_VEL
LIN {X 0,Y 582.588,Z 420.937,A -85,B 0,C 180,E1 25964.035,E2 25964.035} C_VEL
LIN {X 0,Y 570.546,Z 401.354,A -85,B 0,C 180,E1 25962.467,E2 25962.467} C_VEL
LIN {X 0,Y 557.188,Z 381.281,A -85,B 0,C 180,E1 25960.618,E2 25960.618} C_VEL
LIN {X 0,Y 548.562,Z 369.951,A -85,B 0,C 180,E1 25959.37,E2 25959.37} C_VEL
LIN {X 0,Y 545.139,Z 365.328,A -85,B 0,C 180,E1 25958.851,E2 25958.851} C_VEL
LIN {X 0,Y 542.298,Z 361.709,A -85,B 0,C 180,E1 25958.416,E2 25958.416} C_VEL
LIN {X 0,Y 541.197,Z 359.978,A -85,B 0,C 180,E1 25958.238,E2 25958.238} C_VEL
LIN {X 0,Y 538.622,Z 357.309,A -85,B 0,C 180,E1 25957.846,E2 25957.846} C_VEL
LIN {X 0,Y 537.573,Z 354.248,A -85,B 0,C 180,E1 25957.629,E2 25957.629} C_VEL
LIN {X 0,Y 537.62,Z 354.227,A -85,B 0,C 180,E1 25954.301,E2 25954.301} C_VEL
LIN {X 0,Y 537.569,Z 354.256,A -85,B 0,C 180,E1 25951.013,E2 25951.013} C_VEL
LIN {X 0,Y 537.581,Z 354.261,A -85,B 0,C 180,E1 25947.59,E2 25947.59} C_VEL
LIN {X 0,Y 537.617,Z 354.253,A -85,B 0,C 180,E1 25944.27,E2 25944.27} C_VEL
LIN {X 0,Y 537.566,Z 354.256,A -85,B 0,C 180,E1 25940.975,E2 25940.975} C_VEL
LIN {X 0,Y 537.599,Z 354.249,A -85,B 0,C 180,E1 25937.648,E2 25937.648} C_VEL
LIN {X 0,Y 537.575,Z 354.255,A -85,B 0,C 180,E1 25934.543,E2 25934.543} C_VEL
LIN {X 0,Y 537.571,Z 354.263,A -85,B 0,C 180,E1 25931.154,E2 25931.154} C_VEL
LIN {X 0,Y 537.632,Z 354.263,A -85,B 0,C 180,E1 25927.803,E2 25927.803} C_VEL
LIN {X 0,Y 537.571,Z 354.259,A -85,B 0,C 180,E1 25924.463,E2 25924.463} C_VEL
LIN {X 0,Y 537.568,Z 354.251,A -85,B 0,C 180,E1 25920.959,E2 25920.959} C_VEL
LIN {X 0,Y 537.619,Z 354.246,A -85,B 0,C 180,E1 25917.762,E2 25917.762} C_VEL
LIN {X 0,Y 537.566,Z 354.269,A -85,B 0,C 180,E1 25914.45,E2 25914.45} C_VEL
LIN {X 0,Y 537.592,Z 354.266,A -85,B 0,C 180,E1 25911.119,E2 25911.119} C_VEL
LIN {X 0,Y 537.593,Z 354.248,A -85,B 0,C 180,E1 25907.867,E2 25907.867} C_VEL
LIN {X 0,Y 537.562,Z 354.246,A -85,B 0,C 180,E1 25904.574,E2 25904.574} C_VEL
LIN {X 0,Y 537.623,Z 354.245,A -85,B 0,C 180,E1 25901.344,E2 25901.344} C_VEL
LIN {X 0,Y 537.569,Z 354.267,A -85,B 0,C 180,E1 25898.046,E2 25898.046} C_VEL
LIN {X 0,Y 537.571,Z 354.267,A -85,B 0,C 180,E1 25894.554,E2 25894.554} C_VEL
LIN {X 0,Y 537.636,Z 354.264,A -85,B 0,C 180,E1 25891.204,E2 25891.204} C_VEL
LIN {X 0,Y 537.566,Z 354.269,A -85,B 0,C 180,E1 25887.987,E2 25887.987} C_VEL
LIN {X 0,Y 537.581,Z 354.27,A -85,B 0,C 180,E1 25884.555,E2 25884.555} C_VEL
LIN {X 0,Y 537.598,Z 354.432,A -85,B 0,C 180,E1 25882.442,E2 25882.442} C_VEL
LIN {X 0,Y 538.888,Z 357.777,A -85,B 0,C 180,E1 25881.839,E2 25881.839} C_VEL
LIN {X 0,Y 541.452,Z 363.112,A -85,B 0,C 180,E1 25880.834,E2 25880.834} C_VEL
LIN {X 0,Y 545.365,Z 371.859,A -85,B 0,C 180,E1 25879.323,E2 25879.323} C_VEL
LIN {X 0,Y 558.222,Z 390.685,A -85,B 0,C 180,E1 25877.419,E2 25877.419} C_VEL
LIN {X 0,Y 572.345,Z 413.012,A -85,B 0,C 180,E1 25875.471,E2 25875.471} C_VEL
LIN {X 0,Y 582.655,Z 430.952,A -85,B 0,C 180,E1 25874.121,E2 25874.121} C_VEL
LIN {X 0,Y 575.257,Z 689.291,A -85,B 0,C 180,E1 25870.514,E2 25870.514} C_VEL
LIN {X 0,Y 573.021,Z 765.526,A -85,B 0,C 180,E1 25869.436,E2 25869.436} C_VEL
LIN {X 0,Y 571.362,Z 791.034,A -85,B 0,C 180,E1 25868.917,E2 25868.917} C_VEL
LIN {X 0,Y 569.508,Z 813.006,A -85,B 0,C 180,E1 25868.313,E2 25868.313} C_VEL
LIN {X 0,Y 567.08,Z 837.01,A -85,B 0,C 180,E1 25867.468,E2 25867.468} C_VEL
LIN {X 0,Y 564.664,Z 857.615,A -85,B 0,C 180,E1 25866.574,E2 25866.574} C_VEL
LIN {X 0,Y 561.706,Z 880.381,A -85,B 0,C 180,E1 25865.404,E2 25865.404} C_VEL
LIN {X 0,Y 558.718,Z 901.112,A -85,B 0,C 180,E1 25864.128,E2 25864.128} C_VEL
LIN {X 0,Y 555.626,Z 921.636,A -85,B 0,C 180,E1 25862.675,E2 25862.675} C_VEL
LIN {X 0,Y 552.492,Z 941.178,A -85,B 0,C 180,E1 25861.05,E2 25861.05} C_VEL
LIN {X 0,Y 549.706,Z 958.728,A -85,B 0,C 180,E1 25859.392,E2 25859.392} C_VEL
LIN {X 0,Y 546.81,Z 976.686,A -85,B 0,C 180,E1 25857.439,E2 25857.439} C_VEL
LIN {X 0,Y 544.466,Z 991.807,A -85,B 0,C 180,E1 25855.567,E2 25855.567} C_VEL
LIN {X 0,Y 542.061,Z 1008.127,A -85,B 0,C 180,E1 25853.25,E2 25853.25} C_VEL
LIN {X 0,Y 540.311,Z 1021.029,A -85,B 0,C 180,E1 25851.141,E2 25851.141} C_VEL
LIN {X 0,Y 538.643,Z 1034.899,A -85,B 0,C 180,E1 25848.508,E2 25848.508} C_VEL
LIN {X 0,Y 537.634,Z 1044.778,A -85,B 0,C 180,E1 25846.31,E2 25846.31} C_VEL
LIN {X 0,Y 536.807,Z 1054.754,A -85,B 0,C 180,E1 25843.683,E2 25843.683} C_VEL
LIN {X 0,Y 536.35,Z 1061.849,A -85,B 0,C 180,E1 25841.397,E2 25841.397} C_VEL
LIN {X 0,Y 536.065,Z 1068.155,A -85,B 0,C 180,E1 25838.906,E2 25838.906} C_VEL
LIN {X 0,Y 535.95,Z 1072.713,A -85,B 0,C 180,E1 25836.427,E2 25836.427} C_VEL
LIN {X 0,Y 535.918,Z 1075.505,A -85,B 0,C 180,E1 25834.28,E2 25834.28} C_VEL
LIN {X 0,Y 535.906,Z 1077.409,A -85,B 0,C 180,E1 25831.818,E2 25831.818} C_VEL
LIN {X 0,Y 535.906,Z 1077.682,A -85,B 0,C 180,E1 25829.359,E2 25829.359} C_VEL
LIN {X 0,Y 535.915,Z 1076.789,A -85,B 0,C 180,E1 25827.22,E2 25827.22} C_VEL
LIN {X 0,Y 535.934,Z 1074.466,A -85,B 0,C 180,E1 25824.755,E2 25824.755} C_VEL
LIN {X 0,Y 535.99,Z 1070.496,A -85,B 0,C 180,E1 25822.281,E2 25822.281} C_VEL
LIN {X 0,Y 536.155,Z 1065.839,A -85,B 0,C 180,E1 25820.121,E2 25820.121} C_VEL
LIN {X 0,Y 536.526,Z 1058.886,A -85,B 0,C 180,E1 25817.568,E2 25817.568} C_VEL
LIN {X 0,Y 537.135,Z 1050.426,A -85,B 0,C 180,E1 25815.114,E2 25815.114} C_VEL
LIN {X 0,Y 538.052,Z 1040.616,A -85,B 0,C 180,E1 25812.702,E2 25812.702} C_VEL
LIN {X 0,Y 539.349,Z 1028.823,A -85,B 0,C 180,E1 25810.281,E2 25810.281} C_VEL
LIN {X 0,Y 540.915,Z 1016.457,A -85,B 0,C 180,E1 25808.075,E2 25808.075} C_VEL
LIN {X 0,Y 543.014,Z 1001.327,A -85,B 0,C 180,E1 25805.756,E2 25805.756} C_VEL
LIN {X 0,Y 545.091,Z 987.372,A -85,B 0,C 180,E1 25803.881,E2 25803.881} C_VEL
LIN {X 0,Y 547.921,Z 969.064,A -85,B 0,C 180,E1 25801.735,E2 25801.735} C_VEL
LIN {X 0,Y 550.435,Z 952.988,A -85,B 0,C 180,E1 25800.09,E2 25800.09} C_VEL
LIN {X 0,Y 553.61,Z 932.836,A -85,B 0,C 180,E1 25798.287,E2 25798.287} C_VEL
LIN {X 0,Y 556.371,Z 914.575,A -85,B 0,C 180,E1 25796.875,E2 25796.875} C_VEL
LIN {X 0,Y 559.385,Z 894.047,A -85,B 0,C 180,E1 25795.484,E2 25795.484} C_VEL
LIN {X 0,Y 562.224,Z 872.47,A -85,B 0,C 180,E1 25794.252,E2 25794.252} C_VEL
LIN {X 0,Y 564.952,Z 850.686,A -85,B 0,C 180,E1 25793.195,E2 25793.195} C_VEL
LIN {X 0,Y 567.425,Z 827.51,A -85,B 0,C 180,E1 25792.273,E2 25792.273} C_VEL
LIN {X 0,Y 569.383,Z 806.505,A -85,B 0,C 180,E1 25791.595,E2 25791.595} C_VEL
LIN {X 0,Y 571.327,Z 780.859,A -85,B 0,C 180,E1 25790.959,E2 25790.959} C_VEL
LIN {X 0,Y 572.445,Z 758.816,A -85,B 0,C 180,E1 25790.565,E2 25790.565} C_VEL
LIN {X 0,Y 578.81,Z 519.284,A -85,B 0,C 180,E1 25787.25,E2 25787.25} C_VEL
LIN {X 0,Y 581.183,Z 430.246,A -85,B 0,C 180,E1 25786.002,E2 25786.002} C_VEL
LIN {X 0,Y 567.071,Z 405.931,A -85,B 0,C 180,E1 25784.234,E2 25784.234} C_VEL
LIN {X 0,Y 554.721,Z 386.396,A -85,B 0,C 180,E1 25782.598,E2 25782.598} C_VEL
LIN {X 0,Y 546.313,Z 373.784,A -85,B 0,C 180,E1 25781.425,E2 25781.425} C_VEL
LIN {X 0,Y 544.919,Z 371.558,A -85,B 0,C 180,E1 25781.204,E2 25781.204} C_VEL
LIN {X 0,Y 540.498,Z 361.439,A -85,B 0,C 180,E1 25779.518,E2 25779.518} C_VEL
LIN {X 0,Y 538.801,Z 357.546,A -85,B 0,C 180,E1 25778.848,E2 25778.848} C_VEL
LIN {X 0,Y 537.572,Z 354.265,A -85,B 0,C 180,E1 25778.271,E2 25778.271} C_VEL
LIN {X 0,Y 537.62,Z 354.251,A -85,B 0,C 180,E1 25774.948,E2 25774.948} C_VEL
LIN {X 0,Y 537.562,Z 354.258,A -85,B 0,C 180,E1 25771.762,E2 25771.762} C_VEL
LIN {X 0,Y 537.599,Z 354.255,A -85,B 0,C 180,E1 25768.434,E2 25768.434} C_VEL
LIN {X 0,Y 537.588,Z 354.264,A -85,B 0,C 180,E1 25765.21,E2 25765.21} C_VEL
LIN {X 0,Y 537.563,Z 354.266,A -85,B 0,C 180,E1 25761.84,E2 25761.84} C_VEL
LIN {X 0,Y 537.619,Z 354.241,A -85,B 0,C 180,E1 25758.544,E2 25758.544} C_VEL
LIN {X 0,Y 537.569,Z 354.256,A -85,B 0,C 180,E1 25755.315,E2 25755.315} C_VEL
LIN {X 0,Y 537.573,Z 354.267,A -85,B 0,C 180,E1 25751.806,E2 25751.806} C_VEL
LIN {X 0,Y 537.626,Z 354.242,A -85,B 0,C 180,E1 25748.449,E2 25748.449} C_VEL
LIN {X 0,Y 537.565,Z 354.251,A -85,B 0,C 180,E1 25745.229,E2 25745.229} C_VEL
LIN {X 0,Y 537.584,Z 354.268,A -85,B 0,C 180,E1 25741.812,E2 25741.812} C_VEL
LIN {X 0,Y 537.6,Z 354.237,A -85,B 0,C 180,E1 25738.614,E2 25738.614} C_VEL
LIN {X 0,Y 537.564,Z 354.258,A -85,B 0,C 180,E1 25735.306,E2 25735.306} C_VEL
LIN {X 0,Y 537.617,Z 354.259,A -85,B 0,C 180,E1 25731.982,E2 25731.982} C_VEL
LIN {X 0,Y 537.575,Z 354.238,A -85,B 0,C 180,E1 25728.738,E2 25728.738} C_VEL
LIN {X 0,Y 537.569,Z 354.259,A -85,B 0,C 180,E1 25725.287,E2 25725.287} C_VEL
LIN {X 0,Y 537.626,Z 354.257,A -85,B 0,C 180,E1 25722.017,E2 25722.017} C_VEL
LIN {X 0,Y 537.569,Z 354.245,A -85,B 0,C 180,E1 25718.728,E2 25718.728} C_VEL
LIN {X 0,Y 537.585,Z 354.247,A -85,B 0,C 180,E1 25715.378,E2 25715.378} C_VEL
LIN {X 0,Y 537.619,Z 354.263,A -85,B 0,C 180,E1 25712.051,E2 25712.051} C_VEL
LIN {X 0,Y 537.57,Z 354.269,A -85,B 0,C 180,E1 25708.738,E2 25708.738} C_VEL
LIN {X 0,Y 537.607,Z 354.258,A -85,B 0,C 180,E1 25705.44,E2 25705.44} C_VEL
LIN {X 0,Y 537.591,Z 354.263,A -85,B 0,C 180,E1 25702.136,E2 25702.136} C_VEL
LIN {X 0,Y 537.573,Z 354.271,A -85,B 0,C 180,E1 25698.818,E2 25698.818} C_VEL
LIN {X 0,Y 537.651,Z 354.44,A -85,B 0,C 180,E1 25697.56,E2 25697.56} C_VEL
LIN {X 0,Y 538.856,Z 357.626,A -85,B 0,C 180,E1 25697.35,E2 25697.35} C_VEL
LIN {X 0,Y 541.64,Z 360.745,A -85,B 0,C 180,E1 25696.955,E2 25696.955} C_VEL
LIN {X 0,Y 544.3,Z 364.596,A -85,B 0,C 180,E1 25696.567,E2 25696.567} C_VEL
LIN {X 0,Y 545.871,Z 366.544,A -85,B 0,C 180,E1 25696.347,E2 25696.347} C_VEL
LIN {X 0,Y 558.69,Z 384.425,A -85,B 0,C 180,E1 25694.595,E2 25694.595} C_VEL
LIN {X 0,Y 572.771,Z 406.422,A -85,B 0,C 180,E1 25692.778,E2 25692.778} C_VEL
LIN {X 0,Y 581.317,Z 421.073,A -85,B 0,C 180,E1 25691.72,E2 25691.72} C_VEL
LIN {X 0,Y 574.594,Z 667.992,A -85,B 0,C 180,E1 25688.297,E2 25688.297} C_VEL
LIN {X 0,Y 573.08,Z 726.354,A -85,B 0,C 180,E1 25687.495,E2 25687.495} C_VEL
LIN {X 0,Y 572.024,Z 734.039,A -85,B 0,C 180,E1 25687.452,E2 25687.452} C_VEL
LIN {X 0,Y 566.404,Z 753.361,A -85,B 0,C 180,E1 25687.489,E2 25687.489} C_VEL
LIN {X 0,Y 565.216,Z 760.968,A -85,B 0,C 180,E1 25687.394,E2 25687.394} C_VEL
LIN {X 0,Y 563.322,Z 785.096,A -85,B 0,C 180,E1 25686.751,E2 25686.751} C_VEL
LIN {X 0,Y 561.204,Z 807.81,A -85,B 0,C 180,E1 25685.981,E2 25685.981} C_VEL
LIN {X 0,Y 558.613,Z 830.665,A -85,B 0,C 180,E1 25685.007,E2 25685.007} C_VEL
LIN {X 0,Y 556.166,Z 849.641,A -85,B 0,C 180,E1 25684.051,E2 25684.051} C_VEL
LIN {X 0,Y 552.913,Z 872.771,A -85,B 0,C 180,E1 25682.671,E2 25682.671} C_VEL
LIN {X 0,Y 550.056,Z 891.211,A -85,B 0,C 180,E1 25681.38,E2 25681.38} C_VEL
LIN {X 0,Y 546.807,Z 911.299,A -85,B 0,C 180,E1 25679.766,E2 25679.766} C_VEL
LIN {X 0,Y 543.754,Z 929.256,A -85,B 0,C 180,E1 25678.083,E2 25678.083} C_VEL
LIN {X 0,Y 540.822,Z 946.72,A -85,B 0,C 180,E1 25676.223,E2 25676.223} C_VEL
LIN {X 0,Y 538.054,Z 962.697,A -85,B 0,C 180,E1 25674.248,E2 25674.248} C_VEL
LIN {X 0,Y 535.694,Z 977.225,A -85,B 0,C 180,E1 25672.21,E2 25672.21} C_VEL
LIN {X 0,Y 533.393,Z 991.816,A -85,B 0,C 180,E1 25669.834,E2 25669.834} C_VEL
LIN {X 0,Y 531.807,Z 1003.018,A -85,B 0,C 180,E1 25667.733,E2 25667.733} C_VEL
LIN {X 0,Y 530.282,Z 1015.096,A -85,B 0,C 180,E1 25665.083,E2 25665.083} C_VEL
LIN {X 0,Y 529.372,Z 1023.567,A -85,B 0,C 180,E1 25662.878,E2 25662.878} C_VEL
LIN {X 0,Y 528.655,Z 1032.053,A -85,B 0,C 180,E1 25660.241,E2 25660.241} C_VEL
LIN {X 0,Y 528.245,Z 1038.188,A -85,B 0,C 180,E1 25657.833,E2 25657.833} C_VEL
LIN {X 0,Y 528.036,Z 1043.216,A -85,B 0,C 180,E1 25655.324,E2 25655.324} C_VEL
LIN {X 0,Y 527.946,Z 1046.764,A -85,B 0,C 180,E1 25652.714,E2 25652.714} C_VEL
LIN {X 0,Y 527.918,Z 1048.638,A -85,B 0,C 180,E1 25650.434,E2 25650.434} C_VEL
LIN {X 0,Y 527.911,Z 1049.399,A -85,B 0,C 180,E1 25647.829,E2 25647.829} C_VEL
LIN {X 0,Y 527.915,Z 1048.551,A -85,B 0,C 180,E1 25645.328,E2 25645.328} C_VEL
LIN {X 0,Y 527.949,Z 1046.609,A -85,B 0,C 180,E1 25643.038,E2 25643.038} C_VEL
LIN {X 0,Y 528.045,Z 1042.69,A -85,B 0,C 180,E1 25640.298,E2 25640.298} C_VEL
LIN {X 0,Y 528.255,Z 1037.986,A -85,B 0,C 180,E1 25637.983,E2 25637.983} C_VEL
LIN {X 0,Y 528.707,Z 1031.428,A -85,B 0,C 180,E1 25635.432,E2 25635.432} C_VEL
LIN {X 0,Y 529.433,Z 1022.993,A -85,B 0,C 180,E1 25632.865,E2 25632.865} C_VEL
LIN {X 0,Y 530.503,Z 1013.389,A -85,B 0,C 180,E1 25630.397,E2 25630.397} C_VEL
LIN {X 0,Y 532.004,Z 1001.752,A -85,B 0,C 180,E1 25627.909,E2 25627.909} C_VEL
LIN {X 0,Y 533.792,Z 989.652,A -85,B 0,C 180,E1 25625.663,E2 25625.663} C_VEL
LIN {X 0,Y 536.05,Z 975.49,A -85,B 0,C 180,E1 25623.406,E2 25623.406} C_VEL
LIN {X 0,Y 538.508,Z 960.941,A -85,B 0,C 180,E1 25621.377,E2 25621.377} C_VEL
LIN {X 0,Y 541.584,Z 943.283,A -85,B 0,C 180,E1 25619.242,E2 25619.242} C_VEL
LIN {X 0,Y 544.361,Z 927.384,A -85,B 0,C 180,E1 25617.564,E2 25617.564} C_VEL
LIN {X 0,Y 547.94,Z 906.773,A -85,B 0,C 180,E1 25615.676,E2 25615.676} C_VEL
LIN {X 0,Y 550.833,Z 889.337,A -85,B 0,C 180,E1 25614.296,E2 25614.296} C_VEL
LIN {X 0,Y 554.113,Z 868.732,A -85,B 0,C 180,E1 25612.872,E2 25612.872} C_VEL
LIN {X 0,Y 557.021,Z 848.148,A -85,B 0,C 180,E1 25611.67,E2 25611.67} C_VEL
LIN {X 0,Y 559.753,Z 827.581,A -85,B 0,C 180,E1 25610.644,E2 25610.644} C_VEL
LIN {X 0,Y 562.402,Z 803.981,A -85,B 0,C 180,E1 25609.673,E2 25609.673} C_VEL
LIN {X 0,Y 564.454,Z 782.628,A -85,B 0,C 180,E1 25608.964,E2 25608.964} C_VEL
LIN {X 0,Y 566.444,Z 756.724,A -85,B 0,C 180,E1 25608.308,E2 25608.308} C_VEL
LIN {X 0,Y 567.573,Z 734.884,A -85,B 0,C 180,E1 25607.91,E2 25607.91} C_VEL
LIN {X 0,Y 574.974,Z 487.355,A -85,B 0,C 180,E1 25604.425,E2 25604.425} C_VEL
LIN {X 0,Y 576.754,Z 424.351,A -85,B 0,C 180,E1 25603.514,E2 25603.514} C_VEL
LIN {X 0,Y 566.099,Z 406.895,A -85,B 0,C 180,E1 25602.091,E2 25602.091} C_VEL
LIN {X 0,Y 553.282,Z 387.489,A -85,B 0,C 180,E1 25600.28,E2 25600.28} C_VEL
LIN {X 0,Y 544.456,Z 375.833,A -85,B 0,C 180,E1 25598.977,E2 25598.977} C_VEL
LIN {X 0,Y 541.053,Z 371.344,A -85,B 0,C 180,E1 25598.453,E2 25598.453} C_VEL
LIN {X 0,Y 537.278,Z 366.328,A -85,B 0,C 180,E1 25597.856,E2 25597.856} C_VEL
LIN {X 0,Y 534.433,Z 362.708,A -85,B 0,C 180,E1 25597.399,E2 25597.399} C_VEL
LIN {X 0,Y 533.576,Z 361.171,A -85,B 0,C 180,E1 25597.25,E2 25597.25} C_VEL
LIN {X 0,Y 530.914,Z 358.644,A -85,B 0,C 180,E1 25596.829,E2 25596.829} C_VEL
LIN {X 0,Y 529.721,Z 355.604,A -85,B 0,C 180,E1 25596.596,E2 25596.596} C_VEL
LIN {X 0,Y 529.662,Z 355.203,A -85,B 0,C 180,E1 25596.578,E2 25596.578} C_VEL
LIN {X 0,Y 529.628,Z 355.258,A -85,B 0,C 180,E1 25593.244,E2 25593.244} C_VEL
LIN {X 0,Y 529.669,Z 355.254,A -85,B 0,C 180,E1 25589.892,E2 25589.892} C_VEL
LIN {X 0,Y 529.646,Z 355.258,A -85,B 0,C 180,E1 25586.699,E2 25586.699} C_VEL
LIN {X 0,Y 529.631,Z 355.257,A -85,B 0,C 180,E1 25583.239,E2 25583.239} C_VEL
LIN {X 0,Y 529.686,Z 355.254,A -85,B 0,C 180,E1 25579.936,E2 25579.936} C_VEL
LIN {X 0,Y 529.634,Z 355.25,A -85,B 0,C 180,E1 25576.676,E2 25576.676} C_VEL
LIN {X 0,Y 529.631,Z 355.245,A -85,B 0,C 180,E1 25573.205,E2 25573.205} C_VEL
LIN {X 0,Y 529.681,Z 355.233,A -85,B 0,C 180,E1 25569.892,E2 25569.892} C_VEL
LIN {X 0,Y 529.627,Z 355.248,A -85,B 0,C 180,E1 25566.613,E2 25566.613} C_VEL
LIN {X 0,Y 529.638,Z 355.254,A -85,B 0,C 180,E1 25563.138,E2 25563.138} C_VEL
LIN {X 0,Y 529.69,Z 355.247,A -85,B 0,C 180,E1 25559.784,E2 25559.784} C_VEL
LIN {X 0,Y 529.627,Z 355.241,A -85,B 0,C 180,E1 25556.428,E2 25556.428} C_VEL
LIN {X 0,Y 529.634,Z 355.234,A -85,B 0,C 180,E1 25552.951,E2 25552.951} C_VEL
LIN {X 0,Y 529.667,Z 355.242,A -85,B 0,C 180,E1 25549.779,E2 25549.779} C_VEL
LIN {X 0,Y 529.625,Z 355.256,A -85,B 0,C 180,E1 25546.461,E2 25546.461} C_VEL
LIN {X 0,Y 529.669,Z 355.247,A -85,B 0,C 180,E1 25543.156,E2 25543.156} C_VEL
LIN {X 0,Y 529.64,Z 355.236,A -85,B 0,C 180,E1 25539.904,E2 25539.904} C_VEL
LIN {X 0,Y 529.627,Z 355.236,A -85,B 0,C 180,E1 25536.525,E2 25536.525} C_VEL
LIN {X 0,Y 529.683,Z 355.233,A -85,B 0,C 180,E1 25533.238,E2 25533.238} C_VEL
LIN {X 0,Y 529.629,Z 355.255,A -85,B 0,C 180,E1 25529.98,E2 25529.98} C_VEL
LIN {X 0,Y 529.64,Z 355.256,A -85,B 0,C 180,E1 25526.546,E2 25526.546} C_VEL
LIN {X 0,Y 529.685,Z 355.455,A -85,B 0,C 180,E1 25523.424,E2 25523.424} C_VEL
LIN {X 0,Y 531.295,Z 359.193,A -85,B 0,C 180,E1 25522.699,E2 25522.699} C_VEL
LIN {X 0,Y 536.976,Z 371.547,A -85,B 0,C 180,E1 25520.409,E2 25520.409} C_VEL
LIN {X 0,Y 550.839,Z 391.729,A -85,B 0,C 180,E1 25518.261,E2 25518.261} C_VEL
LIN {X 0,Y 562.562,Z 409.865,A -85,B 0,C 180,E1 25516.575,E2 25516.575} C_VEL
LIN {X 0,Y 574.643,Z 430.214,A -85,B 0,C 180,E1 25514.931,E2 25514.931} C_VEL
LIN {X 0,Y 576.866,Z 434.607,A -85,B 0,C 180,E1 25514.631,E2 25514.631} C_VEL
LIN {X 0,Y 569.179,Z 691.344,A -85,B 0,C 180,E1 25511.016,E2 25511.016} C_VEL
LIN {X 0,Y 566.9,Z 765.505,A -85,B 0,C 180,E1 25509.957,E2 25509.957} C_VEL
LIN {X 0,Y 565.176,Z 790.973,A -85,B 0,C 180,E1 25509.434,E2 25509.434} C_VEL
LIN {X 0,Y 563.236,Z 813.045,A -85,B 0,C 180,E1 25508.823,E2 25508.823} C_VEL
LIN {X 0,Y 560.692,Z 837.061,A -85,B 0,C 180,E1 25507.97,E2 25507.97} C_VEL
LIN {X 0,Y 558.175,Z 857.631,A -85,B 0,C 180,E1 25507.07,E2 25507.07} C_VEL
LIN {X 0,Y 555.075,Z 880.433,A -85,B 0,C 180,E1 25505.885,E2 25505.885} C_VEL
LIN {X 0,Y 552.1,Z 900.242,A -85,B 0,C 180,E1 25504.658,E2 25504.658} C_VEL
LIN {X 0,Y 549.066,Z 919.466,A -85,B 0,C 180,E1 25503.293,E2 25503.293} C_VEL
LIN {X 0,Y 545.654,Z 939.851,A -85,B 0,C 180,E1 25501.607,E2 25501.607} C_VEL
LIN {X 0,Y 542.725,Z 957.285,A -85,B 0,C 180,E1 25499.952,E2 25499.952} C_VEL
LIN {X 0,Y 539.48,Z 976.543,A -85,B 0,C 180,E1 25497.844,E2 25497.844} C_VEL
LIN {X 0,Y 536.998,Z 991.652,A -85,B 0,C 180,E1 25495.949,E2 25495.949} C_VEL
LIN {X 0,Y 534.392,Z 1008.386,A -85,B 0,C 180,E1 25493.532,E2 25493.532} C_VEL
LIN {X 0,Y 532.603,Z 1020.77,A -85,B 0,C 180,E1 25491.474,E2 25491.474} C_VEL
LIN {X 0,Y 530.883,Z 1034.172,A -85,B 0,C 180,E1 25488.902,E2 25488.902} C_VEL
LIN {X 0,Y 529.799,Z 1044.095,A -85,B 0,C 180,E1 25486.671,E2 25486.671} C_VEL
LIN {X 0,Y 528.928,Z 1053.815,A -85,B 0,C 180,E1 25484.115,E2 25484.115} C_VEL
LIN {X 0,Y 528.401,Z 1061.322,A -85,B 0,C 180,E1 25481.682,E2 25481.682} C_VEL
LIN {X 0,Y 528.114,Z 1067.163,A -85,B 0,C 180,E1 25479.371,E2 25479.371} C_VEL
LIN {X 0,Y 527.952,Z 1072.334,A -85,B 0,C 180,E1 25476.634,E2 25476.634} C_VEL
LIN {X 0,Y 527.922,Z 1075.175,A -85,B 0,C 180,E1 25474.454,E2 25474.454} C_VEL
LIN {X 0,Y 527.916,Z 1077.058,A -85,B 0,C 180,E1 25472.062,E2 25472.062} C_VEL
LIN {X 0,Y 527.908,Z 1077.492,A -85,B 0,C 180,E1 25469.457,E2 25469.457} C_VEL
LIN {X 0,Y 527.918,Z 1076.576,A -85,B 0,C 180,E1 25467.177,E2 25467.177} C_VEL
LIN {X 0,Y 527.935,Z 1074.252,A -85,B 0,C 180,E1 25464.675,E2 25464.675} C_VEL
LIN {X 0,Y 527.999,Z 1070.282,A -85,B 0,C 180,E1 25462.163,E2 25462.163} C_VEL
LIN {X 0,Y 528.179,Z 1065.365,A -85,B 0,C 180,E1 25459.86,E2 25459.86} C_VEL
LIN {X 0,Y 528.6,Z 1058.139,A -85,B 0,C 180,E1 25457.214,E2 25457.214} C_VEL
LIN {X 0,Y 529.215,Z 1050.208,A -85,B 0,C 180,E1 25454.886,E2 25454.886} C_VEL
LIN {X 0,Y 530.137,Z 1040.857,A -85,B 0,C 180,E1 25452.549,E2 25452.549} C_VEL
LIN {X 0,Y 531.499,Z 1029.162,A -85,B 0,C 180,E1 25450.092,E2 25450.092} C_VEL
LIN {X 0,Y 533.043,Z 1017.489,A -85,B 0,C 180,E1 25447.966,E2 25447.966} C_VEL
LIN {X 0,Y 535.335,Z 1001.832,A -85,B 0,C 180,E1 25445.503,E2 25445.503} C_VEL
LIN {X 0,Y 537.504,Z 987.941,A -85,B 0,C 180,E1 25443.602,E2 25443.602} C_VEL
LIN {X 0,Y 540.38,Z 970.296,A -85,B 0,C 180,E1 25441.485,E2 25441.485} C_VEL
LIN {X 0,Y 543.078,Z 953.791,A -85,B 0,C 180,E1 25439.765,E2 25439.765} C_VEL
LIN {X 0,Y 546.277,Z 934.581,A -85,B 0,C 180,E1 25438.002,E2 25438.002} C_VEL
LIN {X 0,Y 549.333,Z 915.171,A -85,B 0,C 180,E1 25436.476,E2 25436.476} C_VEL
LIN {X 0,Y 552.374,Z 895.308,A -85,B 0,C 180,E1 25435.109,E2 25435.109} C_VEL
LIN {X 0,Y 555.465,Z 873.063,A -85,B 0,C 180,E1 25433.812,E2 25433.812} C_VEL
LIN {X 0,Y 558.076,Z 853.029,A -85,B 0,C 180,E1 25432.822,E2 25432.822} C_VEL
LIN {X 0,Y 560.861,Z 828.542,A -85,B 0,C 180,E1 25431.82,E2 25431.82} C_VEL
LIN {X 0,Y 562.891,Z 807.673,A -85,B 0,C 180,E1 25431.135,E2 25431.135} C_VEL
LIN {X 0,Y 564.894,Z 783.093,A -85,B 0,C 180,E1 25430.504,E2 25430.504} C_VEL
LIN {X 0,Y 566.148,Z 759.815,A -85,B 0,C 180,E1 25430.076,E2 25430.076} C_VEL
LIN {X 0,Y 572.717,Z 523.949,A -85,B 0,C 180,E1 25426.781,E2 25426.781} C_VEL
LIN {X 0,Y 575.229,Z 433.455,A -85,B 0,C 180,E1 25425.5,E2 25425.5} C_VEL
LIN {X 0,Y 561.74,Z 410.227,A -85,B 0,C 180,E1 25423.769,E2 25423.769} C_VEL
LIN {X 0,Y 550.04,Z 391.577,A -85,B 0,C 180,E1 25422.181,E2 25422.181} C_VEL
LIN {X 0,Y 539.44,Z 375.609,A -85,B 0,C 180,E1 25420.657,E2 25420.657} C_VEL
LIN {X 0,Y 536.613,Z 371.19,A -85,B 0,C 180,E1 25420.207,E2 25420.207} C_VEL
LIN {X 0,Y 531.318,Z 359.259,A -85,B 0,C 180,E1 25418.117,E2 25418.117} C_VEL
LIN {X 0,Y 529.841,Z 356.307,A -85,B 0,C 180,E1 25417.557,E2 25417.557} C_VEL
LIN {X 0,Y 529.65,Z 355.241,A -85,B 0,C 180,E1 25417.366,E2 25417.366} C_VEL
LIN {X 0,Y 529.625,Z 355.242,A -85,B 0,C 180,E1 25413.975,E2 25413.975} C_VEL
LIN {X 0,Y 529.678,Z 355.232,A -85,B 0,C 180,E1 25410.643,E2 25410.643} C_VEL
LIN {X 0,Y 529.632,Z 355.234,A -85,B 0,C 180,E1 25407.429,E2 25407.429} C_VEL
LIN {X 0,Y 529.627,Z 355.237,A -85,B 0,C 180,E1 25403.948,E2 25403.948} C_VEL
LIN {X 0,Y 529.688,Z 355.248,A -85,B 0,C 180,E1 25400.671,E2 25400.671} C_VEL
LIN {X 0,Y 529.63,Z 355.253,A -85,B 0,C 180,E1 25397.355,E2 25397.355} C_VEL
LIN {X 0,Y 529.632,Z 355.235,A -85,B 0,C 180,E1 25393.873,E2 25393.873} C_VEL
LIN {X 0,Y 529.679,Z 355.235,A -85,B 0,C 180,E1 25390.551,E2 25390.551} C_VEL
LIN {X 0,Y 529.628,Z 355.256,A -85,B 0,C 180,E1 25387.267,E2 25387.267} C_VEL
LIN {X 0,Y 529.646,Z 355.231,A -85,B 0,C 180,E1 25383.897,E2 25383.897} C_VEL
LIN {X 0,Y 529.662,Z 355.244,A -85,B 0,C 180,E1 25380.649,E2 25380.649} C_VEL
LIN {X 0,Y 529.627,Z 355.256,A -85,B 0,C 180,E1 25377.295,E2 25377.295} C_VEL
LIN {X 0,Y 529.667,Z 355.226,A -85,B 0,C 180,E1 25373.932,E2 25373.932} C_VEL
LIN {X 0,Y 529.638,Z 355.254,A -85,B 0,C 180,E1 25370.766,E2 25370.766} C_VEL
LIN {X 0,Y 529.632,Z 355.248,A -85,B 0,C 180,E1 25367.35,E2 25367.35} C_VEL
LIN {X 0,Y 529.685,Z 355.227,A -85,B 0,C 180,E1 25364.114,E2 25364.114} C_VEL
LIN {X 0,Y 529.631,Z 355.254,A -85,B 0,C 180,E1 25360.822,E2 25360.822} C_VEL
LIN {X 0,Y 529.645,Z 355.254,A -85,B 0,C 180,E1 25357.349,E2 25357.349} C_VEL
LIN {X 0,Y 529.677,Z 355.229,A -85,B 0,C 180,E1 25354.026,E2 25354.026} C_VEL
LIN {X 0,Y 529.628,Z 355.235,A -85,B 0,C 180,E1 25350.727,E2 25350.727} C_VEL
LIN {X 0,Y 529.657,Z 355.238,A -85,B 0,C 180,E1 25347.348,E2 25347.348} C_VEL
LIN {X 0,Y 529.663,Z 355.244,A -85,B 0,C 180,E1 25344.048,E2 25344.048} C_VEL
LIN {X 0,Y 529.629,Z 355.248,A -85,B 0,C 180,E1 25340.718,E2 25340.718} C_VEL
LIN {X 0,Y 529.658,Z 355.461,A -85,B 0,C 180,E1 25338.54,E2 25338.54} C_VEL
LIN {X 0,Y 530.843,Z 358.59,A -85,B 0,C 180,E1 25338.324,E2 25338.324} C_VEL
LIN {X 0,Y 533.807,Z 361.718,A -85,B 0,C 180,E1 25337.888,E2 25337.888} C_VEL
LIN {X 0,Y 536.407,Z 365.576,A -85,B 0,C 180,E1 25337.49,E2 25337.49} C_VEL
LIN {X 0,Y 538.037,Z 367.623,A -85,B 0,C 180,E1 25337.251,E2 25337.251} C_VEL
LIN {X 0,Y 545.712,Z 378.039,A -85,B 0,C 180,E1 25336.145,E2 25336.145} C_VEL
LIN {X 0,Y 556.144,Z 392.807,A -85,B 0,C 180,E1 25334.714,E2 25334.714} C_VEL
LIN {X 0,Y 570.491,Z 415.87,A -85,B 0,C 180,E1 25332.838,E2 25332.838} C_VEL
LIN {X 0,Y 575.39,Z 424.466,A -85,B 0,C 180,E1 25332.219,E2 25332.219} C_VEL
LIN {X 0,Y 568.361,Z 671.373,A -85,B 0,C 180,E1 25328.767,E2 25328.767} C_VEL
LIN {X 0,Y 566.25,Z 742.43,A -85,B 0,C 180,E1 25327.758,E2 25327.758} C_VEL
LIN {X 0,Y 565.216,Z 760.968,A -85,B 0,C 180,E1 25327.394,E2 25327.394} C_VEL
LIN {X 0,Y 563.976,Z 768.571,A -85,B 0,C 180,E1 25327.287,E2 25327.287} C_VEL
LIN {X 0,Y 557.724,Z 787.632,A -85,B 0,C 180,E1 25327.138,E2 25327.138} C_VEL
LIN {X 0,Y 556.189,Z 795.001,A -85,B 0,C 180,E1 25326.952,E2 25326.952} C_VEL
LIN {X 0,Y 553.823,Z 816.925,A -85,B 0,C 180,E1 25326.12,E2 25326.12} C_VEL
LIN {X 0,Y 551.238,Z 837.98,A -85,B 0,C 180,E1 25325.164,E2 25325.164} C_VEL
LIN {X 0,Y 548.084,Z 860.394,A -85,B 0,C 180,E1 25323.935,E2 25323.935} C_VEL
LIN {X 0,Y 545.126,Z 879.682,A -85,B 0,C 180,E1 25322.696,E2 25322.696} C_VEL
LIN {X 0,Y 541.516,Z 901.62,A -85,B 0,C 180,E1 25321.045,E2 25321.045} C_VEL
LIN {X 0,Y 538.535,Z 918.916,A -85,B 0,C 180,E1 25319.536,E2 25319.536} C_VEL
LIN {X 0,Y 535.012,Z 938.668,A -85,B 0,C 180,E1 25317.552,E2 25317.552} C_VEL
LIN {X 0,Y 532.343,Z 953.518,A -85,B 0,C 180,E1 25315.834,E2 25315.834} C_VEL
LIN {X 0,Y 529.529,Z 969.671,A -85,B 0,C 180,E1 25313.716,E2 25313.716} C_VEL
LIN {X 0,Y 527.011,Z 984.287,A -85,B 0,C 180,E1 25311.48,E2 25311.48} C_VEL
LIN {X 0,Y 524.903,Z 997.776,A -85,B 0,C 180,E1 25309.119,E2 25309.119} C_VEL
LIN {X 0,Y 523.254,Z 1009.144,A -85,B 0,C 180,E1 25306.771,E2 25306.771} C_VEL
LIN {X 0,Y 522.018,Z 1019.015,A -85,B 0,C 180,E1 25304.419,E2 25304.419} C_VEL
LIN {X 0,Y 521.073,Z 1027.98,A -85,B 0,C 180,E1 25301.848,E2 25301.848} C_VEL
LIN {X 0,Y 520.512,Z 1034.725,A -85,B 0,C 180,E1 25299.509,E2 25299.509} C_VEL
LIN {X 0,Y 520.15,Z 1040.86,A -85,B 0,C 180,E1 25296.845,E2 25296.845} C_VEL
LIN {X 0,Y 519.998,Z 1044.948,A -85,B 0,C 180,E1 25294.411,E2 25294.411} C_VEL
LIN {X 0,Y 519.945,Z 1047.789,A -85,B 0,C 180,E1 25291.984,E2 25291.984} C_VEL
LIN {X 0,Y 519.924,Z 1049.378,A -85,B 0,C 180,E1 25289.229,E2 25289.229} C_VEL
LIN {X 0,Y 519.92,Z 1049.427,A -85,B 0,C 180,E1 25286.913,E2 25286.913} C_VEL
LIN {X 0,Y 519.94,Z 1048.133,A -85,B 0,C 180,E1 25284.261,E2 25284.261} C_VEL
LIN {X 0,Y 519.999,Z 1045.254,A -85,B 0,C 180,E1 25281.708,E2 25281.708} C_VEL
LIN {X 0,Y 520.127,Z 1041.42,A -85,B 0,C 180,E1 25279.365,E2 25279.365} C_VEL
LIN {X 0,Y 520.489,Z 1035.167,A -85,B 0,C 180,E1 25276.559,E2 25276.559} C_VEL
LIN {X 0,Y 521.042,Z 1028.406,A -85,B 0,C 180,E1 25274.187,E2 25274.187} C_VEL
LIN {X 0,Y 521.993,Z 1019.423,A -85,B 0,C 180,E1 25271.575,E2 25271.575} C_VEL
LIN {X 0,Y 523.276,Z 1009.231,A -85,B 0,C 180,E1 25269.132,E2 25269.132} C_VEL
LIN {X 0,Y 525.083,Z 997.044,A -85,B 0,C 180,E1 25266.614,E2 25266.614} C_VEL
LIN {X 0,Y 527.237,Z 983.565,A -85,B 0,C 180,E1 25264.26,E2 25264.26} C_VEL
LIN {X 0,Y 529.889,Z 968.582,A -85,B 0,C 180,E1 25261.975,E2 25261.975} C_VEL
LIN {X 0,Y 532.701,Z 952.868,A -85,B 0,C 180,E1 25259.918,E2 25259.918} C_VEL
LIN {X 0,Y 535.922,Z 935.701,A -85,B 0,C 180,E1 25257.94,E2 25257.94} C_VEL
LIN {X 0,Y 539.214,Z 917.432,A -85,B 0,C 180,E1 25256.135,E2 25256.135} C_VEL
LIN {X 0,Y 542.562,Z 898.714,A -85,B 0,C 180,E1 25254.513,E2 25254.513} C_VEL
LIN {X 0,Y 546.058,Z 877.896,A -85,B 0,C 180,E1 25252.974,E2 25252.974} C_VEL
LIN {X 0,Y 549.092,Z 858.675,A -85,B 0,C 180,E1 25251.747,E2 25251.747} C_VEL
LIN {X 0,Y 552.425,Z 835.335,A -85,B 0,C 180,E1 25250.49,E2 25250.49} C_VEL
LIN {X 0,Y 554.858,Z 816.079,A -85,B 0,C 180,E1 25249.621,E2 25249.621} C_VEL
LIN {X 0,Y 557.403,Z 793.074,A -85,B 0,C 180,E1 25248.756,E2 25248.756} C_VEL
LIN {X 0,Y 559.415,Z 769.948,A -85,B 0,C 180,E1 25248.084,E2 25248.084} C_VEL
LIN {X 0,Y 560.948,Z 747.908,A -85,B 0,C 180,E1 25247.593,E2 25247.593} C_VEL
LIN {X 0,Y 562.272,Z 713.265,A -85,B 0,C 180,E1 25247.058,E2 25247.058} C_VEL
LIN {X 0,Y 570.153,Z 460.653,A -85,B 0,C 180,E1 25243.479,E2 25243.479} C_VEL
LIN {X 0,Y 571.092,Z 427.886,A -85,B 0,C 180,E1 25242.997,E2 25242.997} C_VEL
LIN {X 0,Y 561.305,Z 411.868,A -85,B 0,C 180,E1 25241.658,E2 25241.658} C_VEL
LIN {X 0,Y 549.264,Z 393.528,A -85,B 0,C 180,E1 25239.919,E2 25239.919} C_VEL
LIN {X 0,Y 537.715,Z 378.063,A -85,B 0,C 180,E1 25238.158,E2 25238.158} C_VEL
LIN {X 0,Y 533.399,Z 372.513,A -85,B 0,C 180,E1 25237.467,E2 25237.467} C_VEL
LIN {X 0,Y 529.57,Z 367.488,A -85,B 0,C 180,E1 25236.833,E2 25236.833} C_VEL
LIN {X 0,Y 526.719,Z 363.943,A -85,B 0,C 180,E1 25236.353,E2 25236.353} C_VEL
LIN {X 0,Y 525.546,Z 362.05,A -85,B 0,C 180,E1 25236.143,E2 25236.143} C_VEL
LIN {X 0,Y 522.876,Z 359.479,A -85,B 0,C 180,E1 25235.696,E2 25235.696} C_VEL
LIN {X 0,Y 521.712,Z 356.383,A -85,B 0,C 180,E1 25235.454,E2 25235.454} C_VEL
LIN {X 0,Y 521.747,Z 356.229,A -85,B 0,C 180,E1 25232.193,E2 25232.193} C_VEL
LIN {X 0,Y 521.692,Z 356.236,A -85,B 0,C 180,E1 25229.007,E2 25229.007} C_VEL
LIN {X 0,Y 521.703,Z 356.229,A -85,B 0,C 180,E1 25225.546,E2 25225.546} C_VEL
LIN {X 0,Y 521.748,Z 356.225,A -85,B 0,C 180,E1 25222.181,E2 25222.181} C_VEL
LIN {X 0,Y 521.69,Z 356.239,A -85,B 0,C 180,E1 25218.9,E2 25218.9} C_VEL
LIN {X 0,Y 521.704,Z 356.242,A -85,B 0,C 180,E1 25215.412,E2 25215.412} C_VEL
LIN {X 0,Y 521.728,Z 356.242,A -85,B 0,C 180,E1 25212.17,E2 25212.17} C_VEL
LIN {X 0,Y 521.686,Z 356.238,A -85,B 0,C 180,E1 25208.82,E2 25208.82} C_VEL
LIN {X 0,Y 521.724,Z 356.222,A -85,B 0,C 180,E1 25205.499,E2 25205.499} C_VEL
LIN {X 0,Y 521.708,Z 356.23,A -85,B 0,C 180,E1 25202.197,E2 25202.197} C_VEL
LIN {X 0,Y 521.689,Z 356.245,A -85,B 0,C 180,E1 25198.792,E2 25198.792} C_VEL
LIN {X 0,Y 521.734,Z 356.243,A -85,B 0,C 180,E1 25195.383,E2 25195.383} C_VEL
LIN {X 0,Y 521.704,Z 356.226,A -85,B 0,C 180,E1 25192.068,E2 25192.068} C_VEL
LIN {X 0,Y 521.685,Z 356.223,A -85,B 0,C 180,E1 25188.614,E2 25188.614} C_VEL
LIN {X 0,Y 521.735,Z 356.222,A -85,B 0,C 180,E1 25185.233,E2 25185.233} C_VEL
LIN {X 0,Y 521.705,Z 356.239,A -85,B 0,C 180,E1 25181.911,E2 25181.911} C_VEL
LIN {X 0,Y 521.689,Z 356.245,A -85,B 0,C 180,E1 25178.526,E2 25178.526} C_VEL
LIN {X 0,Y 521.746,Z 356.234,A -85,B 0,C 180,E1 25175.283,E2 25175.283} C_VEL
LIN {X 0,Y 521.691,Z 356.236,A -85,B 0,C 180,E1 25171.993,E2 25171.993} C_VEL
LIN {X 0,Y 521.693,Z 356.244,A -85,B 0,C 180,E1 25168.45,E2 25168.45} C_VEL
LIN {X 0,Y 521.744,Z 356.239,A -85,B 0,C 180,E1 25165.108,E2 25165.108} C_VEL
LIN {X 0,Y 521.704,Z 356.277,A -85,B 0,C 180,E1 25164.498,E2 25164.498} C_VEL
LIN {X 0,Y 522.774,Z 359.385,A -85,B 0,C 180,E1 25163.907,E2 25163.907} C_VEL
LIN {X 0,Y 523.933,Z 361.432,A -85,B 0,C 180,E1 25163.456,E2 25163.456} C_VEL
LIN {X 0,Y 528.434,Z 371.168,A -85,B 0,C 180,E1 25161.58,E2 25161.58} C_VEL
LIN {X 0,Y 539.128,Z 386.343,A -85,B 0,C 180,E1 25159.822,E2 25159.822} C_VEL
LIN {X 0,Y 550.523,Z 403.277,A -85,B 0,C 180,E1 25158.075,E2 25158.075} C_VEL
LIN {X 0,Y 563.726,Z 424.56,A -85,B 0,C 180,E1 25156.178,E2 25156.178} C_VEL
LIN {X 0,Y 571.142,Z 437.721,A -85,B 0,C 180,E1 25155.158,E2 25155.158} C_VEL
LIN {X 0,Y 563.156,Z 693.159,A -85,B 0,C 180,E1 25151.532,E2 25151.532} C_VEL
LIN {X 0,Y 560.832,Z 765.394,A -85,B 0,C 180,E1 25150.491,E2 25150.491} C_VEL
LIN {X 0,Y 559.048,Z 790.818,A -85,B 0,C 180,E1 25149.965,E2 25149.965} C_VEL
LIN {X 0,Y 557.042,Z 812.768,A -85,B 0,C 180,E1 25149.354,E2 25149.354} C_VEL
LIN {X 0,Y 554.339,Z 837.207,A -85,B 0,C 180,E1 25148.479,E2 25148.479} C_VEL
LIN {X 0,Y 551.734,Z 857.654,A -85,B 0,C 180,E1 25147.577,E2 25147.577} C_VEL
LIN {X 0,Y 548.527,Z 880.226,A -85,B 0,C 180,E1 25146.395,E2 25146.395} C_VEL
LIN {X 0,Y 545.4,Z 900.192,A -85,B 0,C 180,E1 25145.146,E2 25145.146} C_VEL
LIN {X 0,Y 542.016,Z 920.757,A -85,B 0,C 180,E1 25143.666,E2 25143.666} C_VEL
LIN {X 0,Y 538.552,Z 940.361,A -85,B 0,C 180,E1 25142.01,E2 25142.01} C_VEL
LIN {X 0,Y 535.489,Z 957.728,A -85,B 0,C 180,E1 25140.337,E2 25140.337} C_VEL
LIN {X 0,Y 532.179,Z 976.406,A -85,B 0,C 180,E1 25138.26,E2 25138.26} C_VEL
LIN {X 0,Y 529.558,Z 991.503,A -85,B 0,C 180,E1 25136.341,E2 25136.341} C_VEL
LIN {X 0,Y 526.877,Z 1007.787,A -85,B 0,C 180,E1 25133.961,E2 25133.961} C_VEL
LIN {X 0,Y 524.906,Z 1020.594,A -85,B 0,C 180,E1 25131.805,E2 25131.805} C_VEL
LIN {X 0,Y 523.082,Z 1033.981,A -85,B 0,C 180,E1 25129.195,E2 25129.195} C_VEL
LIN {X 0,Y 521.928,Z 1043.894,A -85,B 0,C 180,E1 25126.93,E2 25126.93} C_VEL
LIN {X 0,Y 520.997,Z 1053.602,A -85,B 0,C 180,E1 25124.334,E2 25124.334} C_VEL
LIN {X 0,Y 520.436,Z 1061.105,A -85,B 0,C 180,E1 25121.863,E2 25121.863} C_VEL
LIN {X 0,Y 520.118,Z 1067.204,A -85,B 0,C 180,E1 25119.405,E2 25119.405} C_VEL
LIN {X 0,Y 519.957,Z 1072.119,A -85,B 0,C 180,E1 25116.737,E2 25116.737} C_VEL
LIN {X 0,Y 519.925,Z 1074.96,A -85,B 0,C 180,E1 25114.522,E2 25114.522} C_VEL
LIN {X 0,Y 519.918,Z 1076.844,A -85,B 0,C 180,E1 25112.094,E2 25112.094} C_VEL
LIN {X 0,Y 519.911,Z 1077.278,A -85,B 0,C 180,E1 25109.449,E2 25109.449} C_VEL
LIN {X 0,Y 519.922,Z 1076.363,A -85,B 0,C 180,E1 25107.134,E2 25107.134} C_VEL
LIN {X 0,Y 519.938,Z 1074.038,A -85,B 0,C 180,E1 25104.593,E2 25104.593} C_VEL
LIN {X 0,Y 520.01,Z 1069.984,A -85,B 0,C 180,E1 25101.998,E2 25101.998} C_VEL
LIN {X 0,Y 520.199,Z 1065.15,A -85,B 0,C 180,E1 25099.703,E2 25099.703} C_VEL
LIN {X 0,Y 520.65,Z 1057.92,A -85,B 0,C 180,E1 25097.015,E2 25097.015} C_VEL
LIN {X 0,Y 521.303,Z 1049.98,A -85,B 0,C 180,E1 25094.651,E2 25094.651} C_VEL
LIN {X 0,Y 522.339,Z 1040.151,A -85,B 0,C 180,E1 25092.165,E2 25092.165} C_VEL
LIN {X 0,Y 523.794,Z 1028.323,A -85,B 0,C 180,E1 25089.67,E2 25089.67} C_VEL
LIN {X 0,Y 525.579,Z 1015.933,A -85,B 0,C 180,E1 25087.4,E2 25087.4} C_VEL
LIN {X 0,Y 527.911,Z 1000.767,A -85,B 0,C 180,E1 25085.016,E2 25085.016} C_VEL
LIN {X 0,Y 530.228,Z 986.789,A -85,B 0,C 180,E1 25083.09,E2 25083.09} C_VEL
LIN {X 0,Y 533.358,Z 968.372,A -85,B 0,C 180,E1 25080.882,E2 25080.882} C_VEL
LIN {X 0,Y 536.241,Z 951.777,A -85,B 0,C 180,E1 25079.151,E2 25079.151} C_VEL
LIN {X 0,Y 539.87,Z 930.52,A -85,B 0,C 180,E1 25077.231,E2 25077.231} C_VEL
LIN {X 0,Y 542.847,Z 912.461,A -85,B 0,C 180,E1 25075.82,E2 25075.82} C_VEL
LIN {X 0,Y 546.432,Z 889.637,A -85,B 0,C 180,E1 25074.287,E2 25074.287} C_VEL
LIN {X 0,Y 549.283,Z 869.832,A -85,B 0,C 180,E1 25073.16,E2 25073.16} C_VEL
LIN {X 0,Y 552.341,Z 846.958,A -85,B 0,C 180,E1 25072.057,E2 25072.057} C_VEL
LIN {X 0,Y 554.746,Z 825.697,A -85,B 0,C 180,E1 25071.219,E2 25071.219} C_VEL
LIN {X 0,Y 556.812,Z 805.071,A -85,B 0,C 180,E1 25070.552,E2 25070.552} C_VEL
LIN {X 0,Y 558.849,Z 779.526,A -85,B 0,C 180,E1 25069.919,E2 25069.919} C_VEL
LIN {X 0,Y 560.029,Z 757.601,A -85,B 0,C 180,E1 25069.526,E2 25069.526} C_VEL
LIN {X 0,Y 567.099,Z 514.322,A -85,B 0,C 180,E1 25066.101,E2 25066.101} C_VEL
LIN {X 0,Y 569.298,Z 436.665,A -85,B 0,C 180,E1 25064.986,E2 25064.986} C_VEL
LIN {X 0,Y 555.161,Z 412.311,A -85,B 0,C 180,E1 25063.119,E2 25063.119} C_VEL
LIN {X 0,Y 543.462,Z 393.751,A -85,B 0,C 180,E1 25061.479,E2 25061.479} C_VEL
LIN {X 0,Y 531.779,Z 376.417,A -85,B 0,C 180,E1 25059.739,E2 25059.739} C_VEL
LIN {X 0,Y 527.94,Z 370.718,A -85,B 0,C 180,E1 25059.101,E2 25059.101} C_VEL
LIN {X 0,Y 524.841,Z 363.754,A -85,B 0,C 180,E1 25057.84,E2 25057.84} C_VEL
LIN {X 0,Y 522.901,Z 359.486,A -85,B 0,C 180,E1 25057.038,E2 25057.038} C_VEL
LIN {X 0,Y 521.706,Z 356.235,A -85,B 0,C 180,E1 25056.451,E2 25056.451} C_VEL
LIN {X 0,Y 521.731,Z 356.236,A -85,B 0,C 180,E1 25053.107,E2 25053.107} C_VEL
LIN {X 0,Y 521.686,Z 356.24,A -85,B 0,C 180,E1 25049.745,E2 25049.745} C_VEL
LIN {X 0,Y 521.719,Z 356.226,A -85,B 0,C 180,E1 25046.4,E2 25046.4} C_VEL
LIN {X 0,Y 521.715,Z 356.218,A -85,B 0,C 180,E1 25043.083,E2 25043.083} C_VEL
LIN {X 0,Y 521.685,Z 356.228,A -85,B 0,C 180,E1 25039.714,E2 25039.714} C_VEL
LIN {X 0,Y 521.733,Z 356.241,A -85,B 0,C 180,E1 25036.363,E2 25036.363} C_VEL
LIN {X 0,Y 521.695,Z 356.234,A -85,B 0,C 180,E1 25033.184,E2 25033.184} C_VEL
LIN {X 0,Y 521.689,Z 356.217,A -85,B 0,C 180,E1 25029.71,E2 25029.71} C_VEL
LIN {X 0,Y 521.752,Z 356.237,A -85,B 0,C 180,E1 25026.382,E2 25026.382} C_VEL
LIN {X 0,Y 521.699,Z 356.235,A -85,B 0,C 180,E1 25022.966,E2 25022.966} C_VEL
LIN {X 0,Y 521.69,Z 356.216,A -85,B 0,C 180,E1 25019.561,E2 25019.561} C_VEL
LIN {X 0,Y 521.743,Z 356.242,A -85,B 0,C 180,E1 25016.264,E2 25016.264} C_VEL
LIN {X 0,Y 521.691,Z 356.229,A -85,B 0,C 180,E1 25012.954,E2 25012.954} C_VEL
LIN {X 0,Y 521.696,Z 356.219,A -85,B 0,C 180,E1 25009.49,E2 25009.49} C_VEL
LIN {X 0,Y 521.751,Z 356.241,A -85,B 0,C 180,E1 25006.14,E2 25006.14} C_VEL
LIN {X 0,Y 521.691,Z 356.23,A -85,B 0,C 180,E1 25002.833,E2 25002.833} C_VEL
LIN {X 0,Y 521.7,Z 356.22,A -85,B 0,C 180,E1 24999.35,E2 24999.35} C_VEL
LIN {X 0,Y 521.738,Z 356.235,A -85,B 0,C 180,E1 24996.085,E2 24996.085} C_VEL
LIN {X 0,Y 521.694,Z 356.246,A -85,B 0,C 180,E1 24992.737,E2 24992.737} C_VEL
LIN {X 0,Y 521.715,Z 356.232,A -85,B 0,C 180,E1 24989.349,E2 24989.349} C_VEL
LIN {X 0,Y 521.734,Z 356.225,A -85,B 0,C 180,E1 24985.971,E2 24985.971} C_VEL
LIN {X 0,Y 521.691,Z 356.234,A -85,B 0,C 180,E1 24982.586,E2 24982.586} C_VEL
LIN {X 0,Y 521.778,Z 356.399,A -85,B 0,C 180,E1 24979.558,E2 24979.558} C_VEL
LIN {X 0,Y 522.979,Z 359.628,A -85,B 0,C 180,E1 24979.328,E2 24979.328} C_VEL
LIN {X 0,Y 525.944,Z 362.848,A -85,B 0,C 180,E1 24978.868,E2 24978.868} C_VEL
LIN {X 0,Y 528.492,Z 366.593,A -85,B 0,C 180,E1 24978.46,E2 24978.46} C_VEL
LIN {X 0,Y 530.32,Z 368.719,A -85,B 0,C 180,E1 24978.184,E2 24978.184} C_VEL
LIN {X 0,Y 541.639,Z 384.042,A -85,B 0,C 180,E1 24976.502,E2 24976.502} C_VEL
LIN {X 0,Y 551.99,Z 398.851,A -85,B 0,C 180,E1 24975.052,E2 24975.052} C_VEL
LIN {X 0,Y 565.842,Z 421.277,A -85,B 0,C 180,E1 24973.203,E2 24973.203} C_VEL
LIN {X 0,Y 569.505,Z 427.95,A -85,B 0,C 180,E1 24972.726,E2 24972.726} C_VEL
LIN {X 0,Y 562.193,Z 673.756,A -85,B 0,C 180,E1 24969.261,E2 24969.261} C_VEL
LIN {X 0,Y 560.05,Z 742.763,A -85,B 0,C 180,E1 24968.271,E2 24968.271} C_VEL
LIN {X 0,Y 558.494,Z 767.605,A -85,B 0,C 180,E1 24967.747,E2 24967.747} C_VEL
LIN {X 0,Y 556.702,Z 789.074,A -85,B 0,C 180,E1 24967.143,E2 24967.143} C_VEL
LIN {X 0,Y 556.189,Z 795.001,A -85,B 0,C 180,E1 24966.952,E2 24966.952} C_VEL
LIN {X 0,Y 554.625,Z 802.402,A -85,B 0,C 180,E1 24966.751,E2 24966.751} C_VEL
LIN {X 0,Y 547.803,Z 821.031,A -85,B 0,C 180,E1 24966.409,E2 24966.409} C_VEL
LIN {X 0,Y 546.087,Z 828.142,A -85,B 0,C 180,E1 24966.151,E2 24966.151} C_VEL
LIN {X 0,Y 543.236,Z 848.713,A -85,B 0,C 180,E1 24965.113,E2 24965.113} C_VEL
LIN {X 0,Y 539.955,Z 870.722,A -85,B 0,C 180,E1 24963.802,E2 24963.802} C_VEL
LIN {X 0,Y 536.621,Z 890.593,A -85,B 0,C 180,E1 24962.398,E2 24962.398} C_VEL
LIN {X 0,Y 533.176,Z 910.358,A -85,B 0,C 180,E1 24960.795,E2 24960.795} C_VEL
LIN {X 0,Y 529.69,Z 929.02,A -85,B 0,C 180,E1 24959.021,E2 24959.021} C_VEL
LIN {X 0,Y 526.501,Z 946.269,A -85,B 0,C 180,E1 24957.15,E2 24957.15} C_VEL
LIN {X 0,Y 523.41,Z 962.637,A -85,B 0,C 180,E1 24955.093,E2 24955.093} C_VEL
LIN {X 0,Y 520.952,Z 976.127,A -85,B 0,C 180,E1 24953.165,E2 24953.165} C_VEL
LIN {X 0,Y 518.32,Z 991.274,A -85,B 0,C 180,E1 24950.672,E2 24950.672} C_VEL
LIN {X 0,Y 516.488,Z 1002.577,A -85,B 0,C 180,E1 24948.511,E2 24948.511} C_VEL
LIN {X 0,Y 514.852,Z 1014.038,A -85,B 0,C 180,E1 24945.984,E2 24945.984} C_VEL
LIN {X 0,Y 513.683,Z 1023.402,A -85,B 0,C 180,E1 24943.508,E2 24943.508} C_VEL
LIN {X 0,Y 512.857,Z 1031.735,A -85,B 0,C 180,E1 24940.901,E2 24940.901} C_VEL
LIN {X 0,Y 512.332,Z 1038.256,A -85,B 0,C 180,E1 24938.304,E2 24938.304} C_VEL
LIN {X 0,Y 512.085,Z 1042.948,A -85,B 0,C 180,E1 24935.94,E2 24935.94} C_VEL
LIN {X 0,Y 511.961,Z 1046.921,A -85,B 0,C 180,E1 24933.135,E2 24933.135} C_VEL
LIN {X 0,Y 511.926,Z 1048.902,A -85,B 0,C 180,E1 24930.783,E2 24930.783} C_VEL
LIN {X 0,Y 511.909,Z 1049.755,A -85,B 0,C 180,E1 24928.433,E2 24928.433} C_VEL
LIN {X 0,Y 511.927,Z 1049.208,A -85,B 0,C 180,E1 24925.631,E2 24925.631} C_VEL
LIN {X 0,Y 511.958,Z 1047.422,A -85,B 0,C 180,E1 24923.27,E2 24923.27} C_VEL
LIN {X 0,Y 512.054,Z 1044.168,A -85,B 0,C 180,E1 24920.673,E2 24920.673} C_VEL
LIN {X 0,Y 512.293,Z 1039.036,A -85,B 0,C 180,E1 24917.945,E2 24917.945} C_VEL
LIN {X 0,Y 512.728,Z 1033.212,A -85,B 0,C 180,E1 24915.545,E2 24915.545} C_VEL
LIN {X 0,Y 513.59,Z 1024.442,A -85,B 0,C 180,E1 24912.67,E2 24912.67} C_VEL
LIN {X 0,Y 514.634,Z 1015.897,A -85,B 0,C 180,E1 24910.359,E2 24910.359} C_VEL
LIN {X 0,Y 516.32,Z 1004.278,A -85,B 0,C 180,E1 24907.693,E2 24907.693} C_VEL
LIN {X 0,Y 518.132,Z 992.986,A -85,B 0,C 180,E1 24905.487,E2 24905.487} C_VEL
LIN {X 0,Y 520.574,Z 979.45,A -85,B 0,C 180,E1 24903.168,E2 24903.168} C_VEL
LIN {X 0,Y 523.326,Z 964.419,A -85,B 0,C 180,E1 24900.968,E2 24900.968} C_VEL
LIN {X 0,Y 526.471,Z 948.321,A -85,B 0,C 180,E1 24898.896,E2 24898.896} C_VEL
LIN {X 0,Y 529.883,Z 930.385,A -85,B 0,C 180,E1 24896.912,E2 24896.912} C_VEL
LIN {X 0,Y 533.251,Z 912.846,A -85,B 0,C 180,E1 24895.214,E2 24895.214} C_VEL
LIN {X 0,Y 536.905,Z 892.908,A -85,B 0,C 180,E1 24893.553,E2 24893.553} C_VEL
LIN {X 0,Y 539.99,Z 875.14,A -85,B 0,C 180,E1 24892.267,E2 24892.267} C_VEL
LIN {X 0,Y 543.416,Z 853.979,A -85,B 0,C 180,E1 24890.94,E2 24890.94} C_VEL
LIN {X 0,Y 546.462,Z 832.874,A -85,B 0,C 180,E1 24889.835,E2 24889.835} C_VEL
LIN {X 0,Y 549.328,Z 810.672,A -85,B 0,C 180,E1 24888.852,E2 24888.852} C_VEL
LIN {X 0,Y 551.828,Z 786.94,A -85,B 0,C 180,E1 24888.018,E2 24888.018} C_VEL
LIN {X 0,Y 553.848,Z 764.046,A -85,B 0,C 180,E1 24887.385,E2 24887.385} C_VEL
LIN {X 0,Y 555.383,Z 739.151,A -85,B 0,C 180,E1 24886.892,E2 24886.892} C_VEL
LIN {X 0,Y 563.155,Z 501.688,A -85,B 0,C 180,E1 24883.486,E2 24883.486} C_VEL
LIN {X 0,Y 565.416,Z 431.39,A -85,B 0,C 180,E1 24882.462,E2 24882.462} C_VEL
LIN {X 0,Y 556.326,Z 416.472,A -85,B 0,C 180,E1 24881.185,E2 24881.185} C_VEL
LIN {X 0,Y 545.269,Z 399.555,A -85,B 0,C 180,E1 24879.552,E2 24879.552} C_VEL
LIN {X 0,Y 533.928,Z 384.264,A -85,B 0,C 180,E1 24877.786,E2 24877.786} C_VEL
LIN {X 0,Y 529.276,Z 378.296,A -85,B 0,C 180,E1 24877.026,E2 24877.026} C_VEL
LIN {X 0,Y 525.892,Z 373.843,A -85,B 0,C 180,E1 24876.453,E2 24876.453} C_VEL
LIN {X 0,Y 522.705,Z 369.46,A -85,B 0,C 180,E1 24875.896,E2 24875.896} C_VEL
LIN {X 0,Y 519.096,Z 365.359,A -85,B 0,C 180,E1 24875.267,E2 24875.267} C_VEL
LIN {X 0,Y 517.978,Z 363.279,A -85,B 0,C 180,E1 24875.05,E2 24875.05} C_VEL
LIN {X 0,Y 515.291,Z 360.955,A -85,B 0,C 180,E1 24874.582,E2 24874.582} C_VEL
LIN {X 0,Y 513.906,Z 357.816,A -85,B 0,C 180,E1 24874.291,E2 24874.291} C_VEL
LIN {X 0,Y 513.8,Z 357.19,A -85,B 0,C 180,E1 24874.223,E2 24874.223} C_VEL
LIN {X 0,Y 513.76,Z 357.223,A -85,B 0,C 180,E1 24870.876,E2 24870.876} C_VEL
LIN {X 0,Y 513.755,Z 357.232,A -85,B 0,C 180,E1 24867.343,E2 24867.343} C_VEL
LIN {X 0,Y 513.806,Z 357.223,A -85,B 0,C 180,E1 24863.999,E2 24863.999} C_VEL
LIN {X 0,Y 513.757,Z 357.223,A -85,B 0,C 180,E1 24860.745,E2 24860.745} C_VEL
LIN {X 0,Y 513.752,Z 357.221,A -85,B 0,C 180,E1 24857.207,E2 24857.207} C_VEL
LIN {X 0,Y 513.808,Z 357.209,A -85,B 0,C 180,E1 24853.849,E2 24853.849} C_VEL
LIN {X 0,Y 513.762,Z 357.217,A -85,B 0,C 180,E1 24850.428,E2 24850.428} C_VEL
LIN {X 0,Y 513.751,Z 357.231,A -85,B 0,C 180,E1 24846.931,E2 24846.931} C_VEL
LIN {X 0,Y 513.795,Z 357.231,A -85,B 0,C 180,E1 24843.57,E2 24843.57} C_VEL
LIN {X 0,Y 513.765,Z 357.223,A -85,B 0,C 180,E1 24840.223,E2 24840.223} C_VEL
LIN {X 0,Y 513.747,Z 357.214,A -85,B 0,C 180,E1 24836.764,E2 24836.764} C_VEL
LIN {X 0,Y 513.8,Z 357.208,A -85,B 0,C 180,E1 24833.407,E2 24833.407} C_VEL
LIN {X 0,Y 513.766,Z 357.227,A -85,B 0,C 180,E1 24830.025,E2 24830.025} C_VEL
LIN {X 0,Y 513.749,Z 357.234,A -85,B 0,C 180,E1 24826.608,E2 24826.608} C_VEL
LIN {X 0,Y 513.8,Z 357.219,A -85,B 0,C 180,E1 24823.261,E2 24823.261} C_VEL
LIN {X 0,Y 513.766,Z 357.213,A -85,B 0,C 180,E1 24819.85,E2 24819.85} C_VEL
LIN {X 0,Y 513.747,Z 357.213,A -85,B 0,C 180,E1 24816.447,E2 24816.447} C_VEL
LIN {X 0,Y 513.802,Z 357.209,A -85,B 0,C 180,E1 24813.161,E2 24813.161} C_VEL
LIN {X 0,Y 513.757,Z 357.233,A -85,B 0,C 180,E1 24809.859,E2 24809.859} C_VEL
LIN {X 0,Y 513.751,Z 357.237,A -85,B 0,C 180,E1 24806.311,E2 24806.311} C_VEL
LIN {X 0,Y 513.769,Z 357.249,A -85,B 0,C 180,E1 24805.607,E2 24805.607} C_VEL
LIN {X 0,Y 515.024,Z 360.596,A -85,B 0,C 180,E1 24804.923,E2 24804.923} C_VEL
LIN {X 0,Y 516.063,Z 362.715,A -85,B 0,C 180,E1 24804.461,E2 24804.461} C_VEL
LIN {X 0,Y 520.001,Z 370.822,A -85,B 0,C 180,E1 24802.807,E2 24802.807} C_VEL
LIN {X 0,Y 531.178,Z 386.55,A -85,B 0,C 180,E1 24800.87,E2 24800.87} C_VEL
LIN {X 0,Y 540.135,Z 399.555,A -85,B 0,C 180,E1 24799.423,E2 24799.423} C_VEL
LIN {X 0,Y 552.8,Z 419.25,A -85,B 0,C 180,E1 24797.501,E2 24797.501} C_VEL
LIN {X 0,Y 565.093,Z 440.191,A -85,B 0,C 180,E1 24795.748,E2 24795.748} C_VEL
LIN {X 0,Y 565.446,Z 441.491,A -85,B 0,C 180,E1 24795.687,E2 24795.687} C_VEL
LIN {X 0,Y 557.158,Z 695.623,A -85,B 0,C 180,E1 24792.051,E2 24792.051} C_VEL
LIN {X 0,Y 554.816,Z 765.296,A -85,B 0,C 180,E1 24791.036,E2 24791.036} C_VEL
LIN {X 0,Y 552.972,Z 790.672,A -85,B 0,C 180,E1 24790.507,E2 24790.507} C_VEL
LIN {X 0,Y 550.894,Z 812.588,A -85,B 0,C 180,E1 24789.894,E2 24789.894} C_VEL
LIN {X 0,Y 547.983,Z 837.747,A -85,B 0,C 180,E1 24788.985,E2 24788.985} C_VEL
LIN {X 0,Y 545.336,Z 857.683,A -85,B 0,C 180,E1 24788.096,E2 24788.096} C_VEL
LIN {X 0,Y 541.848,Z 881.103,A -85,B 0,C 180,E1 24786.851,E2 24786.851} C_VEL
LIN {X 0,Y 538.631,Z 900.807,A -85,B 0,C 180,E1 24785.601,E2 24785.601} C_VEL
LIN {X 0,Y 535.089,Z 921.401,A -85,B 0,C 180,E1 24784.097,E2 24784.097} C_VEL
LIN {X 0,Y 531.48,Z 940.876,A -85,B 0,C 180,E1 24782.424,E2 24782.424} C_VEL
LIN {X 0,Y 528.088,Z 959.291,A -85,B 0,C 180,E1 24780.619,E2 24780.619} C_VEL
LIN {X 0,Y 524.731,Z 977.206,A -85,B 0,C 180,E1 24778.574,E2 24778.574} C_VEL
LIN {X 0,Y 521.856,Z 993.063,A -85,B 0,C 180,E1 24776.515,E2 24776.515} C_VEL
LIN {X 0,Y 519.193,Z 1008.334,A -85,B 0,C 180,E1 24774.218,E2 24774.218} C_VEL
LIN {X 0,Y 517.135,Z 1021.066,A -85,B 0,C 180,E1 24772.031,E2 24772.031} C_VEL
LIN {X 0,Y 515.222,Z 1034.319,A -85,B 0,C 180,E1 24769.382,E2 24769.382} C_VEL
LIN {X 0,Y 514.012,Z 1044.168,A -85,B 0,C 180,E1 24767.082,E2 24767.082} C_VEL
LIN {X 0,Y 512.969,Z 1054.477,A -85,B 0,C 180,E1 24764.217,E2 24764.217} C_VEL
LIN {X 0,Y 512.43,Z 1061.513,A -85,B 0,C 180,E1 24761.823,E2 24761.823} C_VEL
LIN {X 0,Y 512.08,Z 1067.948,A -85,B 0,C 180,E1 24759.1,E2 24759.1} C_VEL
LIN {X 0,Y 511.952,Z 1072.229,A -85,B 0,C 180,E1 24756.617,E2 24756.617} C_VEL
LIN {X 0,Y 511.923,Z 1074.977,A -85,B 0,C 180,E1 24754.369,E2 24754.369} C_VEL
LIN {X 0,Y 511.911,Z 1076.831,A -85,B 0,C 180,E1 24751.679,E2 24751.679} C_VEL
LIN {X 0,Y 511.918,Z 1077.019,A -85,B 0,C 180,E1 24749.217,E2 24749.217} C_VEL
LIN {X 0,Y 511.926,Z 1076.08,A -85,B 0,C 180,E1 24746.977,E2 24746.977} C_VEL
LIN {X 0,Y 511.944,Z 1073.538,A -85,B 0,C 180,E1 24744.283,E2 24744.283} C_VEL
LIN {X 0,Y 512.027,Z 1069.641,A -85,B 0,C 180,E1 24741.804,E2 24741.804} C_VEL
LIN {X 0,Y 512.24,Z 1064.67,A -85,B 0,C 180,E1 24739.427,E2 24739.427} C_VEL
LIN {X 0,Y 512.757,Z 1056.97,A -85,B 0,C 180,E1 24736.582,E2 24736.582} C_VEL
LIN {X 0,Y 513.441,Z 1049.328,A -85,B 0,C 180,E1 24734.295,E2 24734.295} C_VEL
LIN {X 0,Y 514.565,Z 1039.422,A -85,B 0,C 180,E1 24731.769,E2 24731.769} C_VEL
LIN {X 0,Y 516.04,Z 1028.059,A -85,B 0,C 180,E1 24729.351,E2 24729.351} C_VEL
LIN {X 0,Y 517.93,Z 1015.659,A -85,B 0,C 180,E1 24727.047,E2 24727.047} C_VEL
LIN {X 0,Y 520.264,Z 1001.259,A -85,B 0,C 180,E1 24724.744,E2 24724.744} C_VEL
LIN {X 0,Y 522.677,Z 987.346,A -85,B 0,C 180,E1 24722.793,E2 24722.793} C_VEL
LIN {X 0,Y 525.97,Z 968.915,A -85,B 0,C 180,E1 24720.538,E2 24720.538} C_VEL
LIN {X 0,Y 528.937,Z 952.57,A -85,B 0,C 180,E1 24718.804,E2 24718.804} C_VEL
LIN {X 0,Y 532.546,Z 932.518,A -85,B 0,C 180,E1 24716.946,E2 24716.946} C_VEL
LIN {X 0,Y 535.794,Z 913.573,A -85,B 0,C 180,E1 24715.436,E2 24715.436} C_VEL
LIN {X 0,Y 539.247,Z 892.861,A -85,B 0,C 180,E1 24714,E2 24714} C_VEL
LIN {X 0,Y 542.496,Z 871.184,A -85,B 0,C 180,E1 24712.738,E2 24712.738} C_VEL
LIN {X 0,Y 545.627,Z 848.934,A -85,B 0,C 180,E1 24711.638,E2 24711.638} C_VEL
LIN {X 0,Y 548.355,Z 825.903,A -85,B 0,C 180,E1 24710.714,E2 24710.714} C_VEL
LIN {X 0,Y 550.466,Z 805.612,A -85,B 0,C 180,E1 24710.05,E2 24710.05} C_VEL
LIN {X 0,Y 552.599,Z 780.143,A -85,B 0,C 180,E1 24709.409,E2 24709.409} C_VEL
LIN {X 0,Y 553.847,Z 757.956,A -85,B 0,C 180,E1 24709.005,E2 24709.005} C_VEL
LIN {X 0,Y 561.199,Z 515.922,A -85,B 0,C 180,E1 24705.566,E2 24705.566} C_VEL
LIN {X 0,Y 563.46,Z 439.96,A -85,B 0,C 180,E1 24704.468,E2 24704.468} C_VEL
LIN {X 0,Y 550.144,Z 416.988,A -85,B 0,C 180,E1 24702.665,E2 24702.665} C_VEL
LIN {X 0,Y 539.004,Z 399.185,A -85,B 0,C 180,E1 24701.066,E2 24701.066} C_VEL
LIN {X 0,Y 527.646,Z 382.254,A -85,B 0,C 180,E1 24699.337,E2 24699.337} C_VEL
LIN {X 0,Y 519.6,Z 370.515,A -85,B 0,C 180,E1 24698.01,E2 24698.01} C_VEL
LIN {X 0,Y 515.191,Z 360.907,A -85,B 0,C 180,E1 24696.158,E2 24696.158} C_VEL
LIN {X 0,Y 513.785,Z 357.398,A -85,B 0,C 180,E1 24695.484,E2 24695.484} C_VEL
LIN {X 0,Y 513.752,Z 357.228,A -85,B 0,C 180,E1 24692.095,E2 24692.095} C_VEL
LIN {X 0,Y 513.814,Z 357.225,A -85,B 0,C 180,E1 24688.856,E2 24688.856} C_VEL
LIN {X 0,Y 513.757,Z 357.232,A -85,B 0,C 180,E1 24685.438,E2 24685.438} C_VEL
LIN {X 0,Y 513.75,Z 357.226,A -85,B 0,C 180,E1 24681.943,E2 24681.943} C_VEL
LIN {X 0,Y 513.802,Z 357.204,A -85,B 0,C 180,E1 24678.607,E2 24678.607} C_VEL
LIN {X 0,Y 513.757,Z 357.217,A -85,B 0,C 180,E1 24675.233,E2 24675.233} C_VEL
LIN {X 0,Y 513.752,Z 357.234,A -85,B 0,C 180,E1 24671.678,E2 24671.678} C_VEL
LIN {X 0,Y 513.8,Z 357.211,A -85,B 0,C 180,E1 24668.28,E2 24668.28} C_VEL
LIN {X 0,Y 513.757,Z 357.21,A -85,B 0,C 180,E1 24665.024,E2 24665.024} C_VEL
LIN {X 0,Y 513.753,Z 357.234,A -85,B 0,C 180,E1 24661.561,E2 24661.561} C_VEL
LIN {X 0,Y 513.804,Z 357.204,A -85,B 0,C 180,E1 24658.216,E2 24658.216} C_VEL
LIN {X 0,Y 513.757,Z 357.214,A -85,B 0,C 180,E1 24654.864,E2 24654.864} C_VEL
LIN {X 0,Y 513.754,Z 357.235,A -85,B 0,C 180,E1 24651.375,E2 24651.375} C_VEL
LIN {X 0,Y 513.799,Z 357.204,A -85,B 0,C 180,E1 24647.981,E2 24647.981} C_VEL
LIN {X 0,Y 513.756,Z 357.217,A -85,B 0,C 180,E1 24644.767,E2 24644.767} C_VEL
LIN {X 0,Y 513.758,Z 357.234,A -85,B 0,C 180,E1 24641.269,E2 24641.269} C_VEL
LIN {X 0,Y 513.814,Z 357.213,A -85,B 0,C 180,E1 24637.866,E2 24637.866} C_VEL
LIN {X 0,Y 513.758,Z 357.208,A -85,B 0,C 180,E1 24634.525,E2 24634.525} C_VEL
LIN {X 0,Y 513.756,Z 357.214,A -85,B 0,C 180,E1 24631.013,E2 24631.013} C_VEL
LIN {X 0,Y 513.805,Z 357.216,A -85,B 0,C 180,E1 24627.645,E2 24627.645} C_VEL
LIN {X 0,Y 513.769,Z 357.226,A -85,B 0,C 180,E1 24624.249,E2 24624.249} C_VEL
LIN {X 0,Y 513.753,Z 357.226,A -85,B 0,C 180,E1 24620.763,E2 24620.763} C_VEL
LIN {X 0,Y 513.784,Z 357.462,A -85,B 0,C 180,E1 24620.644,E2 24620.644} C_VEL
LIN {X 0,Y 514.977,Z 360.579,A -85,B 0,C 180,E1 24620.406,E2 24620.406} C_VEL
LIN {X 0,Y 517.692,Z 363.139,A -85,B 0,C 180,E1 24619.971,E2 24619.971} C_VEL
LIN {X 0,Y 520.579,Z 367.545,A -85,B 0,C 180,E1 24619.482,E2 24619.482} C_VEL
LIN {X 0,Y 522.439,Z 369.688,A -85,B 0,C 180,E1 24619.187,E2 24619.187} C_VEL
LIN {X 0,Y 525.872,Z 374.053,A -85,B 0,C 180,E1 24618.644,E2 24618.644} C_VEL
LIN {X 0,Y 538.036,Z 390.725,A -85,B 0,C 180,E1 24616.796,E2 24616.796} C_VEL
LIN {X 0,Y 547.707,Z 404.638,A -85,B 0,C 180,E1 24615.417,E2 24615.417} C_VEL
LIN {X 0,Y 561.292,Z 426.823,A -85,B 0,C 180,E1 24613.565,E2 24613.565} C_VEL
LIN {X 0,Y 563.671,Z 431.223,A -85,B 0,C 180,E1 24613.247,E2 24613.247} C_VEL
LIN {X 0,Y 556.034,Z 677.254,A -85,B 0,C 180,E1 24609.751,E2 24609.751} C_VEL
LIN {X 0,Y 553.889,Z 743.237,A -85,B 0,C 180,E1 24608.794,E2 24608.794} C_VEL
LIN {X 0,Y 552.273,Z 768.004,A -85,B 0,C 180,E1 24608.265,E2 24608.265} C_VEL
LIN {X 0,Y 550.403,Z 789.611,A -85,B 0,C 180,E1 24607.652,E2 24607.652} C_VEL
LIN {X 0,Y 547.847,Z 813.786,A -85,B 0,C 180,E1 24606.773,E2 24606.773} C_VEL
LIN {X 0,Y 546.087,Z 828.142,A -85,B 0,C 180,E1 24606.151,E2 24606.151} C_VEL
LIN {X 0,Y 544.328,Z 835.328,A -85,B 0,C 180,E1 24605.873,E2 24605.873} C_VEL
LIN {X 0,Y 536.947,Z 853.249,A -85,B 0,C 180,E1 24605.32,E2 24605.32} C_VEL
LIN {X 0,Y 535.072,Z 860.018,A -85,B 0,C 180,E1 24604.984,E2 24604.984} C_VEL
LIN {X 0,Y 531.924,Z 879.096,A -85,B 0,C 180,E1 24603.743,E2 24603.743} C_VEL
LIN {X 0,Y 528.155,Z 900.295,A -85,B 0,C 180,E1 24602.139,E2 24602.139} C_VEL
LIN {X 0,Y 524.745,Z 918.416,A -85,B 0,C 180,E1 24600.539,E2 24600.539} C_VEL
LIN {X 0,Y 521.189,Z 936.989,A -85,B 0,C 180,E1 24598.661,E2 24598.661} C_VEL
LIN {X 0,Y 517.932,Z 953.396,A -85,B 0,C 180,E1 24596.732,E2 24596.732} C_VEL
LIN {X 0,Y 514.808,Z 969.645,A -85,B 0,C 180,E1 24594.56,E2 24594.56} C_VEL
LIN {X 0,Y 512.011,Z 984.313,A -85,B 0,C 180,E1 24592.263,E2 24592.263} C_VEL
LIN {X 0,Y 509.654,Z 997.84,A -85,B 0,C 180,E1 24589.841,E2 24589.841} C_VEL
LIN {X 0,Y 507.692,Z 1009.794,A -85,B 0,C 180,E1 24587.301,E2 24587.301} C_VEL
LIN {X 0,Y 506.265,Z 1020.096,A -85,B 0,C 180,E1 24584.76,E2 24584.76} C_VEL
LIN {X 0,Y 505.212,Z 1028.916,A -85,B 0,C 180,E1 24582.11,E2 24582.11} C_VEL
LIN {X 0,Y 504.592,Z 1035.595,A -85,B 0,C 180,E1 24579.697,E2 24579.697} C_VEL
LIN {X 0,Y 504.172,Z 1041.795,A -85,B 0,C 180,E1 24576.834,E2 24576.834} C_VEL
LIN {X 0,Y 504.013,Z 1045.614,A -85,B 0,C 180,E1 24574.437,E2 24574.437} C_VEL
LIN {X 0,Y 503.947,Z 1048.597,A -85,B 0,C 180,E1 24571.705,E2 24571.705} C_VEL
LIN {X 0,Y 503.93,Z 1049.839,A -85,B 0,C 180,E1 24569.09,E2 24569.09} C_VEL
LIN {X 0,Y 503.926,Z 1049.843,A -85,B 0,C 180,E1 24566.815,E2 24566.815} C_VEL
LIN {X 0,Y 503.953,Z 1048.504,A -85,B 0,C 180,E1 24564.078,E2 24564.078} C_VEL
LIN {X 0,Y 504.014,Z 1045.603,A -85,B 0,C 180,E1 24561.443,E2 24561.443} C_VEL
LIN {X 0,Y 504.178,Z 1041.742,A -85,B 0,C 180,E1 24559.02,E2 24559.02} C_VEL
LIN {X 0,Y 504.618,Z 1035.46,A -85,B 0,C 180,E1 24556.128,E2 24556.128} C_VEL
LIN {X 0,Y 505.228,Z 1029.033,A -85,B 0,C 180,E1 24553.796,E2 24553.796} C_VEL
LIN {X 0,Y 506.311,Z 1020.118,A -85,B 0,C 180,E1 24551.102,E2 24551.102} C_VEL
LIN {X 0,Y 507.714,Z 1010.182,A -85,B 0,C 180,E1 24548.633,E2 24548.633} C_VEL
LIN {X 0,Y 509.527,Z 999.254,A -85,B 0,C 180,E1 24546.279,E2 24546.279} C_VEL
LIN {X 0,Y 511.928,Z 985.82,A -85,B 0,C 180,E1 24543.805,E2 24543.805} C_VEL
LIN {X 0,Y 514.478,Z 972.616,A -85,B 0,C 180,E1 24541.692,E2 24541.692} C_VEL
LIN {X 0,Y 517.843,Z 955.761,A -85,B 0,C 180,E1 24539.353,E2 24539.353} C_VEL
LIN {X 0,Y 520.978,Z 940.319,A -85,B 0,C 180,E1 24537.494,E2 24537.494} C_VEL
LIN {X 0,Y 524.868,Z 921.068,A -85,B 0,C 180,E1 24535.476,E2 24535.476} C_VEL
LIN {X 0,Y 528.307,Z 903.339,A -85,B 0,C 180,E1 24533.875,E2 24533.875} C_VEL
LIN {X 0,Y 532.095,Z 883.218,A -85,B 0,C 180,E1 24532.291,E2 24532.291} C_VEL
LIN {X 0,Y 535.572,Z 862.977,A -85,B 0,C 180,E1 24530.943,E2 24530.943} C_VEL
LIN {X 0,Y 538.989,Z 841.653,A -85,B 0,C 180,E1 24529.721,E2 24529.721} C_VEL
LIN {X 0,Y 542.071,Z 819.471,A -85,B 0,C 180,E1 24528.673,E2 24528.673} C_VEL
LIN {X 0,Y 544.441,Z 799.917,A -85,B 0,C 180,E1 24527.899,E2 24527.899} C_VEL
LIN {X 0,Y 546.964,Z 775.211,A -85,B 0,C 180,E1 24527.117,E2 24527.117} C_VEL
LIN {X 0,Y 548.613,Z 753.902,A -85,B 0,C 180,E1 24526.608,E2 24526.608} C_VEL
LIN {X 0,Y 549.906,Z 729.728,A -85,B 0,C 180,E1 24526.18,E2 24526.18} C_VEL
LIN {X 0,Y 558.448,Z 476.825,A -85,B 0,C 180,E1 24522.54,E2 24522.54} C_VEL
LIN {X 0,Y 559.794,Z 434.861,A -85,B 0,C 180,E1 24521.915,E2 24521.915} C_VEL
LIN {X 0,Y 548.365,Z 416.204,A -85,B 0,C 180,E1 24520.254,E2 24520.254} C_VEL
LIN {X 0,Y 539.659,Z 403.371,A -85,B 0,C 180,E1 24518.928,E2 24518.928} C_VEL
